LIN {X 104.584,Y 102.598,Z 81.000,A 180.000,B 0.000,C 180.000} C_DIS
LIN {X 104.698,Y 102.438,Z 81.000,A 180.000,B 0.000,C 180.000} C_DIS
LIN {X 104.762,Y 102.341,Z 81.000,A 180.000,B 0.000,C 180.000} C_DIS
LIN {X 104.817,Y 102.260,Z 81.000,A 180.000,B 0.000,C 180.000} C_DIS
LIN {X 104.931,Y 102.081,Z 81.000,A 180.000,B 0.000,C 180.000} C_DIS
LIN {X 105.036,Y 101.902,Z 81.000,A 180.000,B 0.000,C 180.000} C_DIS
LIN {X 105.120,Y 101.755,Z 81.000,A 180.000,B 0.000,C 180.000} C_DIS
LIN {X 105.137,Y 101.723,Z 81.000,A 180.000,B 0.000,C 180.000} C_DIS
LIN {X 105.234,Y 101.545,Z 81.000,A 180.000,B 0.000,C 180.000} C_DIS
LIN {X 105.326,Y 101.366,Z 81.000,A 180.000,B 0.000,C 180.000} C_DIS
LIN {X 105.413,Y 101.187,Z 81.000,A 180.000,B 0.000,C 180.000} C_DIS
LIN {X 105.493,Y 101.008,Z 81.000,A 180.000,B 0.000,C 180.000} C_DIS
LIN {X 105.568,Y 100.829,Z 81.000,A 180.000,B 0.000,C 180.000} C_DIS
LIN {X 105.638,Y 100.651,Z 81.000,A 180.000,B 0.000,C 180.000} C_DIS
LIN {X 105.706,Y 100.472,Z 81.000,A 180.000,B 0.000,C 180.000} C_DIS
LIN {X 105.771,Y 100.293,Z 81.000,A 180.000,B 0.000,C 180.000} C_DIS
LIN {X 105.835,Y 100.092,Z 81.000,A 180.000,B 0.000,C 180.000} C_DIS
LIN {X 105.883,Y 99.936,Z 81.000,A 180.000,B 0.000,C 180.000} C_DIS
LIN {X 105.929,Y 99.757,Z 81.000,A 180.000,B 0.000,C 180.000} C_DIS
LIN {X 105.975,Y 99.578,Z 81.000,A 180.000,B 0.000,C 180.000} C_DIS
LIN {X 106.014,Y 99.427,Z 81.000,A 180.000,B 0.000,C 180.000} C_DIS
LIN {X 106.020,Y 99.399,Z 81.000,A 180.000,B 0.000,C 180.000} C_DIS
LIN {X 106.057,Y 99.221,Z 81.000,A 180.000,B 0.000,C 180.000} C_DIS
LIN {X 106.093,Y 99.042,Z 81.000,A 180.000,B 0.000,C 180.000} C_DIS
LIN {X 106.121,Y 98.863,Z 81.000,A 180.000,B 0.000,C 180.000} C_DIS
LIN {X 106.146,Y 98.684,Z 81.000,A 180.000,B 0.000,C 180.000} C_DIS
LIN {X 106.169,Y 98.505,Z 81.000,A 180.000,B 0.000,C 180.000} C_DIS
LIN {X 106.190,Y 98.327,Z 81.000,A 180.000,B 0.000,C 180.000} C_DIS
LIN {X 106.205,Y 98.148,Z 81.000,A 180.000,B 0.000,C 180.000} C_DIS
LIN {X 106.218,Y 97.969,Z 81.000,A 180.000,B 0.000,C 180.000} C_DIS
LIN {X 106.223,Y 97.790,Z 81.000,A 180.000,B 0.000,C 180.000} C_DIS
LIN {X 106.227,Y 97.612,Z 81.000,A 180.000,B 0.000,C 180.000} C_DIS
LIN {X 106.227,Y 97.433,Z 81.000,A 180.000,B 0.000,C 180.000} C_DIS
LIN {X 106.224,Y 97.254,Z 81.000,A 180.000,B 0.000,C 180.000} C_DIS
LIN {X 106.219,Y 97.075,Z 81.000,A 180.000,B 0.000,C 180.000} C_DIS
LIN {X 106.208,Y 96.897,Z 81.000,A 180.000,B 0.000,C 180.000} C_DIS
LIN {X 106.193,Y 96.709,Z 81.000,A 180.000,B 0.000,C 180.000} C_DIS
LIN {X 106.175,Y 96.539,Z 81.000,A 180.000,B 0.000,C 180.000} C_DIS
LIN {X 106.152,Y 96.360,Z 81.000,A 180.000,B 0.000,C 180.000} C_DIS
LIN {X 106.127,Y 96.181,Z 81.000,A 180.000,B 0.000,C 180.000} C_DIS
LIN {X 106.101,Y 96.003,Z 81.000,A 180.000,B 0.000,C 180.000} C_DIS
LIN {X 106.066,Y 95.824,Z 81.000,A 180.000,B 0.000,C 180.000} C_DIS
LIN {X 106.030,Y 95.645,Z 81.000,A 180.000,B 0.000,C 180.000} C_DIS
LIN {X 106.014,Y 95.573,Z 81.000,A 180.000,B 0.000,C 180.000} C_DIS
LIN {X 105.987,Y 95.466,Z 81.000,A 180.000,B 0.000,C 180.000} C_DIS
LIN {X 105.941,Y 95.288,Z 81.000,A 180.000,B 0.000,C 180.000} C_DIS
LIN {X 105.894,Y 95.109,Z 81.000,A 180.000,B 0.000,C 180.000} C_DIS
LIN {X 105.842,Y 94.930,Z 81.000,A 180.000,B 0.000,C 180.000} C_DIS
LIN {X 105.785,Y 94.751,Z 81.000,A 180.000,B 0.000,C 180.000} C_DIS
LIN {X 105.723,Y 94.573,Z 81.000,A 180.000,B 0.000,C 180.000} C_DIS
LIN {X 105.655,Y 94.394,Z 81.000,A 180.000,B 0.000,C 180.000} C_DIS
LIN {X 105.585,Y 94.215,Z 81.000,A 180.000,B 0.000,C 180.000} C_DIS
LIN {X 105.512,Y 94.036,Z 81.000,A 180.000,B 0.000,C 180.000} C_DIS
LIN {X 105.477,Y 93.958,Z 81.000,A 180.000,B 0.000,C 180.000} C_DIS
LIN {X 105.432,Y 93.857,Z 81.000,A 180.000,B 0.000,C 180.000} C_DIS
LIN {X 105.349,Y 93.679,Z 81.000,A 180.000,B 0.000,C 180.000} C_DIS
LIN {X 105.299,Y 93.581,Z 81.000,A 180.000,B 0.000,C 180.000} C_DIS
LIN {X 105.257,Y 93.500,Z 81.000,A 180.000,B 0.000,C 180.000} C_DIS
LIN {X 105.162,Y 93.321,Z 81.000,A 180.000,B 0.000,C 180.000} C_DIS
LIN {X 105.120,Y 93.245,Z 81.000,A 180.000,B 0.000,C 180.000} C_DIS
LIN {X 105.063,Y 93.142,Z 81.000,A 180.000,B 0.000,C 180.000} C_DIS
LIN {X 104.941,Y 92.936,Z 81.000,A 180.000,B 0.000,C 180.000} C_DIS
LIN {X 104.847,Y 92.785,Z 81.000,A 180.000,B 0.000,C 180.000} C_DIS
LIN {X 104.727,Y 92.606,Z 81.000,A 180.000,B 0.000,C 180.000} C_DIS
LIN {X 104.602,Y 92.427,Z 81.000,A 180.000,B 0.000,C 180.000} C_DIS
LIN {X 104.584,Y 92.402,Z 81.000,A 180.000,B 0.000,C 180.000} C_DIS
LIN {X 104.470,Y 92.249,Z 81.000,A 180.000,B 0.000,C 180.000} C_DIS
LIN {X 104.405,Y 92.162,Z 81.000,A 180.000,B 0.000,C 180.000} C_DIS
LIN {X 104.335,Y 92.070,Z 81.000,A 180.000,B 0.000,C 180.000} C_DIS
LIN {X 104.226,Y 91.936,Z 81.000,A 180.000,B 0.000,C 180.000} C_DIS
LIN {X 104.188,Y 91.891,Z 81.000,A 180.000,B 0.000,C 180.000} C_DIS
LIN {X 104.047,Y 91.726,Z 81.000,A 180.000,B 0.000,C 180.000} C_DIS
LIN {X 104.035,Y 91.712,Z 81.000,A 180.000,B 0.000,C 180.000} C_DIS
LIN {X 103.869,Y 91.535,Z 81.000,A 180.000,B 0.000,C 180.000} C_DIS
LIN {X 103.690,Y 91.346,Z 81.000,A 180.000,B 0.000,C 180.000} C_DIS
LIN {X 103.516,Y 91.176,Z 81.000,A 180.000,B 0.000,C 180.000} C_DIS
LIN {X 103.511,Y 91.171,Z 81.000,A 180.000,B 0.000,C 180.000} C_DIS
LIN {X 103.332,Y 91.004,Z 81.000,A 180.000,B 0.000,C 180.000} C_DIS
LIN {X 103.324,Y 90.997,Z 81.000,A 180.000,B 0.000,C 180.000} C_DIS
LIN {X 103.153,Y 90.852,Z 81.000,A 180.000,B 0.000,C 180.000} C_DIS
LIN {X 103.113,Y 90.818,Z 81.000,A 180.000,B 0.000,C 180.000} C_DIS
LIN {X 102.975,Y 90.703,Z 81.000,A 180.000,B 0.000,C 180.000} C_DIS
LIN {X 102.897,Y 90.640,Z 81.000,A 180.000,B 0.000,C 180.000} C_DIS
LIN {X 102.796,Y 90.562,Z 81.000,A 180.000,B 0.000,C 180.000} C_DIS
LIN {X 102.662,Y 90.461,Z 81.000,A 180.000,B 0.000,C 180.000} C_DIS
LIN {X 102.617,Y 90.427,Z 81.000,A 180.000,B 0.000,C 180.000} C_DIS
LIN {X 102.438,Y 90.303,Z 81.000,A 180.000,B 0.000,C 180.000} C_DIS
LIN {X 102.407,Y 90.282,Z 81.000,A 180.000,B 0.000,C 180.000} C_DIS
LIN {X 102.260,Y 90.184,Z 81.000,A 180.000,B 0.000,C 180.000} C_DIS
LIN {X 102.132,Y 90.103,Z 81.000,A 180.000,B 0.000,C 180.000} C_DIS
LIN {X 102.081,Y 90.071,Z 81.000,A 180.000,B 0.000,C 180.000} C_DIS
LIN {X 101.902,Y 89.963,Z 81.000,A 180.000,B 0.000,C 180.000} C_DIS
LIN {X 101.836,Y 89.925,Z 81.000,A 180.000,B 0.000,C 180.000} C_DIS
LIN {X 101.723,Y 89.859,Z 81.000,A 180.000,B 0.000,C 180.000} C_DIS
LIN {X 101.545,Y 89.765,Z 81.000,A 180.000,B 0.000,C 180.000} C_DIS
LIN {X 101.506,Y 89.746,Z 81.000,A 180.000,B 0.000,C 180.000} C_DIS
LIN {X 101.366,Y 89.674,Z 81.000,A 180.000,B 0.000,C 180.000} C_DIS
LIN {X 101.187,Y 89.590,Z 81.000,A 180.000,B 0.000,C 180.000} C_DIS
LIN {X 101.138,Y 89.567,Z 81.000,A 180.000,B 0.000,C 180.000} C_DIS
LIN {X 101.008,Y 89.509,Z 81.000,A 180.000,B 0.000,C 180.000} C_DIS
LIN {X 100.829,Y 89.430,Z 81.000,A 180.000,B 0.000,C 180.000} C_DIS
LIN {X 100.725,Y 89.388,Z 81.000,A 180.000,B 0.000,C 180.000} C_DIS
LIN {X 100.651,Y 89.360,Z 81.000,A 180.000,B 0.000,C 180.000} C_DIS
LIN {X 100.472,Y 89.292,Z 81.000,A 180.000,B 0.000,C 180.000} C_DIS
LIN {X 100.293,Y 89.232,Z 81.000,A 180.000,B 0.000,C 180.000} C_DIS
LIN {X 100.223,Y 89.209,Z 81.000,A 180.000,B 0.000,C 180.000} C_DIS
LIN {X 100.114,Y 89.175,Z 81.000,A 180.000,B 0.000,C 180.000} C_DIS
LIN {X 99.936,Y 89.118,Z 81.000,A 180.000,B 0.000,C 180.000} C_DIS
LIN {X 99.757,Y 89.068,Z 81.000,A 180.000,B 0.000,C 180.000} C_DIS
LIN {X 99.578,Y 89.022,Z 81.000,A 180.000,B 0.000,C 180.000} C_DIS
LIN {X 99.399,Y 88.981,Z 81.000,A 180.000,B 0.000,C 180.000} C_DIS
LIN {X 99.221,Y 88.945,Z 81.000,A 180.000,B 0.000,C 180.000} C_DIS
LIN {X 99.042,Y 88.910,Z 81.000,A 180.000,B 0.000,C 180.000} C_DIS
LIN {X 98.863,Y 88.878,Z 81.000,A 180.000,B 0.000,C 180.000} C_DIS
LIN {X 98.682,Y 88.852,Z 81.000,A 180.000,B 0.000,C 180.000} C_DIS
LIN {X 98.505,Y 88.828,Z 81.000,A 180.000,B 0.000,C 180.000} C_DIS
LIN {X 98.327,Y 88.811,Z 81.000,A 180.000,B 0.000,C 180.000} C_DIS
LIN {X 98.148,Y 88.796,Z 81.000,A 180.000,B 0.000,C 180.000} C_DIS
LIN {X 97.969,Y 88.785,Z 81.000,A 180.000,B 0.000,C 180.000} C_DIS
LIN {X 97.790,Y 88.777,Z 81.000,A 180.000,B 0.000,C 180.000} C_DIS
LIN {X 97.612,Y 88.772,Z 81.000,A 180.000,B 0.000,C 180.000} C_DIS
LIN {X 97.433,Y 88.770,Z 81.000,A 180.000,B 0.000,C 180.000} C_DIS
LIN {X 97.254,Y 88.775,Z 81.000,A 180.000,B 0.000,C 180.000} C_DIS
LIN {X 97.075,Y 88.782,Z 81.000,A 180.000,B 0.000,C 180.000} C_DIS
LIN {X 96.897,Y 88.793,Z 81.000,A 180.000,B 0.000,C 180.000} C_DIS
LIN {X 96.718,Y 88.808,Z 81.000,A 180.000,B 0.000,C 180.000} C_DIS
LIN {X 96.539,Y 88.823,Z 81.000,A 180.000,B 0.000,C 180.000} C_DIS
LIN {X 96.360,Y 88.846,Z 81.000,A 180.000,B 0.000,C 180.000} C_DIS
LIN {X 96.181,Y 88.871,Z 81.000,A 180.000,B 0.000,C 180.000} C_DIS
LIN {X 96.003,Y 88.902,Z 81.000,A 180.000,B 0.000,C 180.000} C_DIS
LIN {X 95.824,Y 88.936,Z 81.000,A 180.000,B 0.000,C 180.000} C_DIS
LIN {X 95.645,Y 88.972,Z 81.000,A 180.000,B 0.000,C 180.000} C_DIS
LIN {X 95.466,Y 89.010,Z 81.000,A 180.000,B 0.000,C 180.000} C_DIS
LIN {X 95.387,Y 89.031,Z 81.000,A 180.000,B 0.000,C 180.000} C_DIS
LIN {X 95.288,Y 89.056,Z 81.000,A 180.000,B 0.000,C 180.000} C_DIS
LIN {X 95.109,Y 89.104,Z 81.000,A 180.000,B 0.000,C 180.000} C_DIS
LIN {X 94.930,Y 89.161,Z 81.000,A 180.000,B 0.000,C 180.000} C_DIS
LIN {X 94.777,Y 89.209,Z 81.000,A 180.000,B 0.000,C 180.000} C_DIS
LIN {X 94.751,Y 89.218,Z 81.000,A 180.000,B 0.000,C 180.000} C_DIS
LIN {X 94.573,Y 89.276,Z 81.000,A 180.000,B 0.000,C 180.000} C_DIS
LIN {X 94.394,Y 89.343,Z 81.000,A 180.000,B 0.000,C 180.000} C_DIS
LIN {X 94.275,Y 89.388,Z 81.000,A 180.000,B 0.000,C 180.000} C_DIS
LIN {X 94.215,Y 89.411,Z 81.000,A 180.000,B 0.000,C 180.000} C_DIS
LIN {X 94.036,Y 89.489,Z 81.000,A 180.000,B 0.000,C 180.000} C_DIS
LIN {X 93.862,Y 89.567,Z 81.000,A 180.000,B 0.000,C 180.000} C_DIS
LIN {X 93.857,Y 89.569,Z 81.000,A 180.000,B 0.000,C 180.000} C_DIS
LIN {X 93.679,Y 89.653,Z 81.000,A 180.000,B 0.000,C 180.000} C_DIS
LIN {X 93.500,Y 89.742,Z 81.000,A 180.000,B 0.000,C 180.000} C_DIS
LIN {X 93.321,Y 89.835,Z 81.000,A 180.000,B 0.000,C 180.000} C_DIS
LIN {X 93.164,Y 89.925,Z 81.000,A 180.000,B 0.000,C 180.000} C_DIS
LIN {X 93.142,Y 89.937,Z 81.000,A 180.000,B 0.000,C 180.000} C_DIS
LIN {X 92.964,Y 90.043,Z 81.000,A 180.000,B 0.000,C 180.000} C_DIS
LIN {X 92.868,Y 90.103,Z 81.000,A 180.000,B 0.000,C 180.000} C_DIS
LIN {X 92.785,Y 90.156,Z 81.000,A 180.000,B 0.000,C 180.000} C_DIS
LIN {X 92.606,Y 90.274,Z 81.000,A 180.000,B 0.000,C 180.000} C_DIS
LIN {X 92.593,Y 90.282,Z 81.000,A 180.000,B 0.000,C 180.000} C_DIS
LIN {X 92.427,Y 90.395,Z 81.000,A 180.000,B 0.000,C 180.000} C_DIS
LIN {X 92.338,Y 90.461,Z 81.000,A 180.000,B 0.000,C 180.000} C_DIS
LIN {X 92.249,Y 90.528,Z 81.000,A 180.000,B 0.000,C 180.000} C_DIS
LIN {X 92.103,Y 90.640,Z 81.000,A 180.000,B 0.000,C 180.000} C_DIS
LIN {X 92.070,Y 90.667,Z 81.000,A 180.000,B 0.000,C 180.000} C_DIS
LIN {X 91.891,Y 90.815,Z 81.000,A 180.000,B 0.000,C 180.000} C_DIS
LIN {X 91.712,Y 90.966,Z 81.000,A 180.000,B 0.000,C 180.000} C_DIS
LIN {X 91.676,Y 90.997,Z 81.000,A 180.000,B 0.000,C 180.000} C_DIS
LIN {X 91.533,Y 91.129,Z 81.000,A 180.000,B 0.000,C 180.000} C_DIS
LIN {X 91.484,Y 91.176,Z 81.000,A 180.000,B 0.000,C 180.000} C_DIS
LIN {X 91.355,Y 91.300,Z 81.000,A 180.000,B 0.000,C 180.000} C_DIS
LIN {X 91.302,Y 91.355,Z 81.000,A 180.000,B 0.000,C 180.000} C_DIS
LIN {X 91.133,Y 91.533,Z 81.000,A 180.000,B 0.000,C 180.000} C_DIS
LIN {X 90.997,Y 91.678,Z 81.000,A 180.000,B 0.000,C 180.000} C_DIS
LIN {X 90.965,Y 91.712,Z 81.000,A 180.000,B 0.000,C 180.000} C_DIS
LIN {X 90.818,Y 91.884,Z 81.000,A 180.000,B 0.000,C 180.000} C_DIS
LIN {X 90.812,Y 91.891,Z 81.000,A 180.000,B 0.000,C 180.000} C_DIS
LIN {X 90.665,Y 92.070,Z 81.000,A 180.000,B 0.000,C 180.000} C_DIS
LIN {X 90.640,Y 92.103,Z 81.000,A 180.000,B 0.000,C 180.000} C_DIS
LIN {X 90.530,Y 92.249,Z 81.000,A 180.000,B 0.000,C 180.000} C_DIS
LIN {X 90.461,Y 92.341,Z 81.000,A 180.000,B 0.000,C 180.000} C_DIS
LIN {X 90.398,Y 92.427,Z 81.000,A 180.000,B 0.000,C 180.000} C_DIS
LIN {X 90.282,Y 92.592,Z 81.000,A 180.000,B 0.000,C 180.000} C_DIS
LIN {X 90.153,Y 92.785,Z 81.000,A 180.000,B 0.000,C 180.000} C_DIS
LIN {X 90.103,Y 92.862,Z 81.000,A 180.000,B 0.000,C 180.000} C_DIS
LIN {X 90.082,Y 92.898,Z 81.000,A 180.000,B 0.000,C 180.000} C_DIS
; Link Move Starts
LIN {X 89.924,Y 93.166,Z 81.000,A 180.000,B 0.000,C 180.000} C_DIS
LIN {X 89.783,Y 93.422,Z 80.999,A 180.000,B 0.000,C 180.000} C_DIS
LIN {X 89.639,Y 93.700,Z 80.998,A 180.000,B 0.000,C 180.000} C_DIS
LIN {X 89.518,Y 93.964,Z 80.996,A 180.000,B 0.000,C 180.000} C_DIS
LIN {X 89.405,Y 94.233,Z 80.995,A 180.000,B 0.000,C 180.000} C_DIS
LIN {X 89.292,Y 94.523,Z 80.992,A 180.000,B 0.000,C 180.000} C_DIS
LIN {X 89.195,Y 94.796,Z 80.989,A 180.000,B 0.000,C 180.000} C_DIS
LIN {X 89.108,Y 95.073,Z 80.986,A 180.000,B 0.000,C 180.000} C_DIS
LIN {X 89.028,Y 95.376,Z 80.983,A 180.000,B 0.000,C 180.000} C_DIS
LIN {X 88.956,Y 95.663,Z 80.979,A 180.000,B 0.000,C 180.000} C_DIS
LIN {X 88.896,Y 95.955,Z 80.974,A 180.000,B 0.000,C 180.000} C_DIS
LIN {X 88.849,Y 96.249,Z 80.970,A 180.000,B 0.000,C 180.000} C_DIS
LIN {X 88.827,Y 96.403,Z 80.967,A 180.000,B 0.000,C 180.000} C_DIS
LIN {X 88.806,Y 96.556,Z 80.965,A 180.000,B 0.000,C 180.000} C_DIS
LIN {X 88.790,Y 96.704,Z 80.962,A 180.000,B 0.000,C 180.000} C_DIS
LIN {X 88.776,Y 96.852,Z 80.959,A 180.000,B 0.000,C 180.000} C_DIS
LIN {X 88.764,Y 96.996,Z 80.957,A 180.000,B 0.000,C 180.000} C_DIS
LIN {X 88.757,Y 97.141,Z 80.954,A 180.000,B 0.000,C 180.000} C_DIS
LIN {X 88.752,Y 97.292,Z 80.951,A 180.000,B 0.000,C 180.000} C_DIS
LIN {X 88.748,Y 97.443,Z 80.948,A 180.000,B 0.000,C 180.000} C_DIS
LIN {X 88.747,Y 97.595,Z 80.944,A 180.000,B 0.000,C 180.000} C_DIS
LIN {X 88.748,Y 97.747,Z 80.941,A 180.000,B 0.000,C 180.000} C_DIS
LIN {X 88.751,Y 97.896,Z 80.938,A 180.000,B 0.000,C 180.000} C_DIS
LIN {X 88.756,Y 98.044,Z 80.934,A 180.000,B 0.000,C 180.000} C_DIS
LIN {X 88.767,Y 98.194,Z 80.931,A 180.000,B 0.000,C 180.000} C_DIS
LIN {X 88.778,Y 98.344,Z 80.927,A 180.000,B 0.000,C 180.000} C_DIS
LIN {X 88.793,Y 98.492,Z 80.924,A 180.000,B 0.000,C 180.000} C_DIS
LIN {X 88.810,Y 98.640,Z 80.920,A 180.000,B 0.000,C 180.000} C_DIS
LIN {X 88.830,Y 98.796,Z 80.916,A 180.000,B 0.000,C 180.000} C_DIS
LIN {X 88.850,Y 98.951,Z 80.912,A 180.000,B 0.000,C 180.000} C_DIS
LIN {X 88.874,Y 99.095,Z 80.908,A 180.000,B 0.000,C 180.000} C_DIS
LIN {X 88.901,Y 99.239,Z 80.904,A 180.000,B 0.000,C 180.000} C_DIS
LIN {X 88.928,Y 99.382,Z 80.900,A 180.000,B 0.000,C 180.000} C_DIS
LIN {X 88.961,Y 99.525,Z 80.896,A 180.000,B 0.000,C 180.000} C_DIS
LIN {X 88.998,Y 99.677,Z 80.892,A 180.000,B 0.000,C 180.000} C_DIS
LIN {X 89.036,Y 99.830,Z 80.888,A 180.000,B 0.000,C 180.000} C_DIS
LIN {X 89.071,Y 99.972,Z 80.883,A 180.000,B 0.000,C 180.000} C_DIS
LIN {X 89.112,Y 100.113,Z 80.879,A 180.000,B 0.000,C 180.000} C_DIS
LIN {X 89.156,Y 100.255,Z 80.875,A 180.000,B 0.000,C 180.000} C_DIS
LIN {X 89.200,Y 100.397,Z 80.870,A 180.000,B 0.000,C 180.000} C_DIS
LIN {X 89.253,Y 100.541,Z 80.865,A 180.000,B 0.000,C 180.000} C_DIS
LIN {X 89.305,Y 100.685,Z 80.861,A 180.000,B 0.000,C 180.000} C_DIS
LIN {X 89.358,Y 100.824,Z 80.856,A 180.000,B 0.000,C 180.000} C_DIS
LIN {X 89.412,Y 100.964,Z 80.851,A 180.000,B 0.000,C 180.000} C_DIS
LIN {X 89.473,Y 101.106,Z 80.846,A 180.000,B 0.000,C 180.000} C_DIS
LIN {X 89.503,Y 101.176,Z 80.844,A 180.000,B 0.000,C 180.000} C_DIS
LIN {X 89.533,Y 101.247,Z 80.841,A 180.000,B 0.000,C 180.000} C_DIS
LIN {X 89.596,Y 101.381,Z 80.836,A 180.000,B 0.000,C 180.000} C_DIS
LIN {X 89.662,Y 101.514,Z 80.831,A 180.000,B 0.000,C 180.000} C_DIS
LIN {X 89.696,Y 101.582,Z 80.829,A 180.000,B 0.000,C 180.000} C_DIS
LIN {X 89.730,Y 101.650,Z 80.826,A 180.000,B 0.000,C 180.000} C_DIS
LIN {X 89.765,Y 101.717,Z 80.824,A 180.000,B 0.000,C 180.000} C_DIS
LIN {X 89.801,Y 101.784,Z 80.821,A 180.000,B 0.000,C 180.000} C_DIS
LIN {X 89.836,Y 101.851,Z 80.818,A 180.000,B 0.000,C 180.000} C_DIS
LIN {X 89.873,Y 101.918,Z 80.816,A 180.000,B 0.000,C 180.000} C_DIS
LIN {X 89.949,Y 102.051,Z 80.811,A 180.000,B 0.000,C 180.000} C_DIS
LIN {X 89.985,Y 102.115,Z 80.808,A 180.000,B 0.000,C 180.000} C_DIS
LIN {X 90.022,Y 102.178,Z 80.805,A 180.000,B 0.000,C 180.000} C_DIS
LIN {X 90.060,Y 102.241,Z 80.803,A 180.000,B 0.000,C 180.000} C_DIS
LIN {X 90.100,Y 102.303,Z 80.800,A 180.000,B 0.000,C 180.000} C_DIS
LIN {X 90.183,Y 102.431,Z 80.795,A 180.000,B 0.000,C 180.000} C_DIS
LIN {X 90.224,Y 102.496,Z 80.792,A 180.000,B 0.000,C 180.000} C_DIS
LIN {X 90.267,Y 102.559,Z 80.790,A 180.000,B 0.000,C 180.000} C_DIS
LIN {X 90.354,Y 102.683,Z 80.784,A 180.000,B 0.000,C 180.000} C_DIS
LIN {X 90.398,Y 102.745,Z 80.782,A 180.000,B 0.000,C 180.000} C_DIS
LIN {X 90.443,Y 102.807,Z 80.779,A 180.000,B 0.000,C 180.000} C_DIS
LIN {X 90.532,Y 102.929,Z 80.774,A 180.000,B 0.000,C 180.000} C_DIS
LIN {X 90.576,Y 102.991,Z 80.771,A 180.000,B 0.000,C 180.000} C_DIS
LIN {X 90.622,Y 103.051,Z 80.768,A 180.000,B 0.000,C 180.000} C_DIS
LIN {X 90.669,Y 103.109,Z 80.766,A 180.000,B 0.000,C 180.000} C_DIS
LIN {X 90.764,Y 103.225,Z 80.761,A 180.000,B 0.000,C 180.000} C_DIS
LIN {X 90.812,Y 103.283,Z 80.758,A 180.000,B 0.000,C 180.000} C_DIS
LIN {X 90.860,Y 103.342,Z 80.755,A 180.000,B 0.000,C 180.000} C_DIS
LIN {X 90.910,Y 103.398,Z 80.753,A 180.000,B 0.000,C 180.000} C_DIS
LIN {X 91.012,Y 103.510,Z 80.747,A 180.000,B 0.000,C 180.000} C_DIS
LIN {X 91.065,Y 103.568,Z 80.745,A 180.000,B 0.000,C 180.000} C_DIS
LIN {X 91.171,Y 103.684,Z 80.739,A 180.000,B 0.000,C 180.000} C_DIS
LIN {X 91.224,Y 103.742,Z 80.736,A 180.000,B 0.000,C 180.000} C_DIS
LIN {X 91.275,Y 103.796,Z 80.734,A 180.000,B 0.000,C 180.000} C_DIS
LIN {X 91.327,Y 103.848,Z 80.731,A 180.000,B 0.000,C 180.000} C_DIS
LIN {X 91.486,Y 104.004,Z 80.724,A 180.000,B 0.000,C 180.000} C_DIS
LIN {X 91.539,Y 104.055,Z 80.721,A 180.000,B 0.000,C 180.000} C_DIS
LIN {X 91.594,Y 104.106,Z 80.718,A 180.000,B 0.000,C 180.000} C_DIS
LIN {X 91.649,Y 104.154,Z 80.716,A 180.000,B 0.000,C 180.000} C_DIS
LIN {X 91.767,Y 104.257,Z 80.710,A 180.000,B 0.000,C 180.000} C_DIS
LIN {X 91.825,Y 104.308,Z 80.708,A 180.000,B 0.000,C 180.000} C_DIS
LIN {X 91.884,Y 104.359,Z 80.705,A 180.000,B 0.000,C 180.000} C_DIS
LIN {X 91.942,Y 104.408,Z 80.702,A 180.000,B 0.000,C 180.000} C_DIS
LIN {X 91.999,Y 104.456,Z 80.700,A 180.000,B 0.000,C 180.000} C_DIS
LIN {X 92.057,Y 104.504,Z 80.697,A 180.000,B 0.000,C 180.000} C_DIS
LIN {X 92.116,Y 104.550,Z 80.694,A 180.000,B 0.000,C 180.000} C_DIS
LIN {X 92.236,Y 104.644,Z 80.689,A 180.000,B 0.000,C 180.000} C_DIS
LIN {X 92.296,Y 104.691,Z 80.686,A 180.000,B 0.000,C 180.000} C_DIS
LIN {X 92.357,Y 104.737,Z 80.684,A 180.000,B 0.000,C 180.000} C_DIS
LIN {X 92.419,Y 104.780,Z 80.681,A 180.000,B 0.000,C 180.000} C_DIS
LIN {X 92.543,Y 104.866,Z 80.676,A 180.000,B 0.000,C 180.000} C_DIS
LIN {X 92.605,Y 104.909,Z 80.673,A 180.000,B 0.000,C 180.000} C_DIS
LIN {X 92.669,Y 104.953,Z 80.670,A 180.000,B 0.000,C 180.000} C_DIS
LIN {X 92.733,Y 104.995,Z 80.668,A 180.000,B 0.000,C 180.000} C_DIS
LIN {X 92.797,Y 105.037,Z 80.665,A 180.000,B 0.000,C 180.000} C_DIS
LIN {X 92.861,Y 105.079,Z 80.662,A 180.000,B 0.000,C 180.000} C_DIS
LIN {X 92.925,Y 105.119,Z 80.660,A 180.000,B 0.000,C 180.000} C_DIS
LIN {X 93.119,Y 105.237,Z 80.652,A 180.000,B 0.000,C 180.000} C_DIS
LIN {X 93.184,Y 105.277,Z 80.649,A 180.000,B 0.000,C 180.000} C_DIS
LIN {X 93.251,Y 105.314,Z 80.647,A 180.000,B 0.000,C 180.000} C_DIS
LIN {X 93.318,Y 105.351,Z 80.644,A 180.000,B 0.000,C 180.000} C_DIS
LIN {X 93.453,Y 105.423,Z 80.639,A 180.000,B 0.000,C 180.000} C_DIS
LIN {X 93.520,Y 105.459,Z 80.636,A 180.000,B 0.000,C 180.000} C_DIS
LIN {X 93.588,Y 105.493,Z 80.633,A 180.000,B 0.000,C 180.000} C_DIS
LIN {X 93.725,Y 105.561,Z 80.628,A 180.000,B 0.000,C 180.000} C_DIS
LIN {X 93.795,Y 105.595,Z 80.625,A 180.000,B 0.000,C 180.000} C_DIS
LIN {X 94.003,Y 105.692,Z 80.617,A 180.000,B 0.000,C 180.000} C_DIS
LIN {X 94.071,Y 105.723,Z 80.615,A 180.000,B 0.000,C 180.000} C_DIS
LIN {X 94.139,Y 105.753,Z 80.612,A 180.000,B 0.000,C 180.000} C_DIS
LIN {X 94.209,Y 105.781,Z 80.609,A 180.000,B 0.000,C 180.000} C_DIS
LIN {X 94.420,Y 105.866,Z 80.601,A 180.000,B 0.000,C 180.000} C_DIS
LIN {X 94.491,Y 105.893,Z 80.599,A 180.000,B 0.000,C 180.000} C_DIS
LIN {X 94.564,Y 105.919,Z 80.596,A 180.000,B 0.000,C 180.000} C_DIS
LIN {X 94.711,Y 105.970,Z 80.591,A 180.000,B 0.000,C 180.000} C_DIS
LIN {X 94.785,Y 105.995,Z 80.588,A 180.000,B 0.000,C 180.000} C_DIS
LIN {X 95.002,Y 106.068,Z 80.580,A 180.000,B 0.000,C 180.000} C_DIS
LIN {X 95.075,Y 106.091,Z 80.577,A 180.000,B 0.000,C 180.000} C_DIS
LIN {X 95.148,Y 106.113,Z 80.574,A 180.000,B 0.000,C 180.000} C_DIS
LIN {X 95.368,Y 106.173,Z 80.567,A 180.000,B 0.000,C 180.000} C_DIS
LIN {X 95.442,Y 106.193,Z 80.564,A 180.000,B 0.000,C 180.000} C_DIS
LIN {X 95.516,Y 106.211,Z 80.561,A 180.000,B 0.000,C 180.000} C_DIS
LIN {X 95.590,Y 106.227,Z 80.559,A 180.000,B 0.000,C 180.000} C_DIS
LIN {X 95.817,Y 106.276,Z 80.550,A 180.000,B 0.000,C 180.000} C_DIS
LIN {X 95.894,Y 106.292,Z 80.548,A 180.000,B 0.000,C 180.000} C_DIS
LIN {X 95.970,Y 106.308,Z 80.545,A 180.000,B 0.000,C 180.000} C_DIS
LIN {X 96.045,Y 106.323,Z 80.542,A 180.000,B 0.000,C 180.000} C_DIS
LIN {X 96.119,Y 106.337,Z 80.540,A 180.000,B 0.000,C 180.000} C_DIS
LIN {X 96.194,Y 106.349,Z 80.537,A 180.000,B 0.000,C 180.000} C_DIS
LIN {X 96.343,Y 106.372,Z 80.532,A 180.000,B 0.000,C 180.000} C_DIS
LIN {X 96.418,Y 106.384,Z 80.529,A 180.000,B 0.000,C 180.000} C_DIS
LIN {X 96.493,Y 106.394,Z 80.526,A 180.000,B 0.000,C 180.000} C_DIS
LIN {X 96.567,Y 106.402,Z 80.524,A 180.000,B 0.000,C 180.000} C_DIS
LIN {X 96.801,Y 106.426,Z 80.516,A 180.000,B 0.000,C 180.000} C_DIS
LIN {X 96.879,Y 106.433,Z 80.513,A 180.000,B 0.000,C 180.000} C_DIS
LIN {X 97.031,Y 106.445,Z 80.508,A 180.000,B 0.000,C 180.000} C_DIS
LIN {X 97.107,Y 106.451,Z 80.505,A 180.000,B 0.000,C 180.000} C_DIS
LIN {X 97.183,Y 106.455,Z 80.502,A 180.000,B 0.000,C 180.000} C_DIS
LIN {X 97.412,Y 106.465,Z 80.494,A 180.000,B 0.000,C 180.000} C_DIS
LIN {X 97.489,Y 106.468,Z 80.492,A 180.000,B 0.000,C 180.000} C_DIS
LIN {X 97.566,Y 106.468,Z 80.489,A 180.000,B 0.000,C 180.000} C_DIS
LIN {X 97.796,Y 106.465,Z 80.481,A 180.000,B 0.000,C 180.000} C_DIS
LIN {X 97.874,Y 106.464,Z 80.478,A 180.000,B 0.000,C 180.000} C_DIS
LIN {X 97.951,Y 106.461,Z 80.475,A 180.000,B 0.000,C 180.000} C_DIS
LIN {X 98.106,Y 106.454,Z 80.470,A 180.000,B 0.000,C 180.000} C_DIS
LIN {X 98.183,Y 106.450,Z 80.467,A 180.000,B 0.000,C 180.000} C_DIS
LIN {X 98.415,Y 106.434,Z 80.459,A 180.000,B 0.000,C 180.000} C_DIS
LIN {X 98.491,Y 106.429,Z 80.457,A 180.000,B 0.000,C 180.000} C_DIS
LIN {X 98.567,Y 106.421,Z 80.454,A 180.000,B 0.000,C 180.000} C_DIS
LIN {X 98.642,Y 106.412,Z 80.451,A 180.000,B 0.000,C 180.000} C_DIS
LIN {X 98.868,Y 106.384,Z 80.443,A 180.000,B 0.000,C 180.000} C_DIS
LIN {X 98.944,Y 106.373,Z 80.441,A 180.000,B 0.000,C 180.000} C_DIS
LIN {X 99.019,Y 106.361,Z 80.438,A 180.000,B 0.000,C 180.000} C_DIS
LIN {X 99.174,Y 106.334,Z 80.432,A 180.000,B 0.000,C 180.000} C_DIS
LIN {X 99.251,Y 106.320,Z 80.430,A 180.000,B 0.000,C 180.000} C_DIS
LIN {X 99.478,Y 106.279,Z 80.422,A 180.000,B 0.000,C 180.000} C_DIS
LIN {X 99.553,Y 106.264,Z 80.419,A 180.000,B 0.000,C 180.000} C_DIS
LIN {X 99.627,Y 106.247,Z 80.416,A 180.000,B 0.000,C 180.000} C_DIS
LIN {X 99.851,Y 106.193,Z 80.408,A 180.000,B 0.000,C 180.000} C_DIS
LIN {X 99.926,Y 106.174,Z 80.406,A 180.000,B 0.000,C 180.000} C_DIS
LIN {X 100.001,Y 106.154,Z 80.403,A 180.000,B 0.000,C 180.000} C_DIS
LIN {X 100.075,Y 106.131,Z 80.400,A 180.000,B 0.000,C 180.000} C_DIS
LIN {X 100.224,Y 106.086,Z 80.395,A 180.000,B 0.000,C 180.000} C_DIS
LIN {X 100.299,Y 106.064,Z 80.392,A 180.000,B 0.000,C 180.000} C_DIS
LIN {X 100.447,Y 106.018,Z 80.387,A 180.000,B 0.000,C 180.000} C_DIS
LIN {X 100.522,Y 105.995,Z 80.384,A 180.000,B 0.000,C 180.000} C_DIS
LIN {X 100.595,Y 105.970,Z 80.381,A 180.000,B 0.000,C 180.000} C_DIS
LIN {X 100.740,Y 105.918,Z 80.376,A 180.000,B 0.000,C 180.000} C_DIS
LIN {X 100.812,Y 105.891,Z 80.373,A 180.000,B 0.000,C 180.000} C_DIS
LIN {X 100.884,Y 105.865,Z 80.370,A 180.000,B 0.000,C 180.000} C_DIS
LIN {X 100.956,Y 105.837,Z 80.368,A 180.000,B 0.000,C 180.000} C_DIS
LIN {X 101.026,Y 105.807,Z 80.365,A 180.000,B 0.000,C 180.000} C_DIS
LIN {X 101.168,Y 105.747,Z 80.360,A 180.000,B 0.000,C 180.000} C_DIS
LIN {X 101.240,Y 105.716,Z 80.357,A 180.000,B 0.000,C 180.000} C_DIS
LIN {X 101.311,Y 105.685,Z 80.354,A 180.000,B 0.000,C 180.000} C_DIS
LIN {X 101.452,Y 105.621,Z 80.349,A 180.000,B 0.000,C 180.000} C_DIS
LIN {X 101.522,Y 105.589,Z 80.346,A 180.000,B 0.000,C 180.000} C_DIS
LIN {X 101.592,Y 105.555,Z 80.343,A 180.000,B 0.000,C 180.000} C_DIS
LIN {X 101.661,Y 105.520,Z 80.341,A 180.000,B 0.000,C 180.000} C_DIS
LIN {X 101.799,Y 105.452,Z 80.335,A 180.000,B 0.000,C 180.000} C_DIS
LIN {X 101.868,Y 105.417,Z 80.333,A 180.000,B 0.000,C 180.000} C_DIS
LIN {X 101.936,Y 105.379,Z 80.330,A 180.000,B 0.000,C 180.000} C_DIS
LIN {X 102.070,Y 105.303,Z 80.325,A 180.000,B 0.000,C 180.000} C_DIS
LIN {X 102.137,Y 105.265,Z 80.322,A 180.000,B 0.000,C 180.000} C_DIS
LIN {X 102.205,Y 105.226,Z 80.319,A 180.000,B 0.000,C 180.000} C_DIS
LIN {X 102.271,Y 105.186,Z 80.316,A 180.000,B 0.000,C 180.000} C_DIS
LIN {X 102.404,Y 105.105,Z 80.311,A 180.000,B 0.000,C 180.000} C_DIS
LIN {X 102.470,Y 105.063,Z 80.308,A 180.000,B 0.000,C 180.000} C_DIS
LIN {X 102.600,Y 104.980,Z 80.303,A 180.000,B 0.000,C 180.000} C_DIS
LIN {X 102.665,Y 104.938,Z 80.300,A 180.000,B 0.000,C 180.000} C_DIS
LIN {X 102.729,Y 104.896,Z 80.298,A 180.000,B 0.000,C 180.000} C_DIS
LIN {X 102.794,Y 104.851,Z 80.295,A 180.000,B 0.000,C 180.000} C_DIS
LIN {X 102.857,Y 104.806,Z 80.292,A 180.000,B 0.000,C 180.000} C_DIS
LIN {X 103.046,Y 104.668,Z 80.284,A 180.000,B 0.000,C 180.000} C_DIS
LIN {X 103.107,Y 104.622,Z 80.281,A 180.000,B 0.000,C 180.000} C_DIS
LIN {X 103.168,Y 104.573,Z 80.279,A 180.000,B 0.000,C 180.000} C_DIS
LIN {X 103.229,Y 104.525,Z 80.276,A 180.000,B 0.000,C 180.000} C_DIS
LIN {X 103.290,Y 104.476,Z 80.273,A 180.000,B 0.000,C 180.000} C_DIS
LIN {X 103.350,Y 104.427,Z 80.270,A 180.000,B 0.000,C 180.000} C_DIS
LIN {X 103.471,Y 104.328,Z 80.265,A 180.000,B 0.000,C 180.000} C_DIS
LIN {X 103.531,Y 104.279,Z 80.262,A 180.000,B 0.000,C 180.000} C_DIS
LIN {X 103.590,Y 104.229,Z 80.259,A 180.000,B 0.000,C 180.000} C_DIS
LIN {X 103.647,Y 104.177,Z 80.257,A 180.000,B 0.000,C 180.000} C_DIS
LIN {X 103.704,Y 104.125,Z 80.254,A 180.000,B 0.000,C 180.000} C_DIS
LIN {X 103.818,Y 104.021,Z 80.249,A 180.000,B 0.000,C 180.000} C_DIS
LIN {X 103.875,Y 103.968,Z 80.246,A 180.000,B 0.000,C 180.000} C_DIS
LIN {X 103.930,Y 103.914,Z 80.243,A 180.000,B 0.000,C 180.000} C_DIS
LIN {X 103.985,Y 103.858,Z 80.241,A 180.000,B 0.000,C 180.000} C_DIS
LIN {X 104.094,Y 103.745,Z 80.235,A 180.000,B 0.000,C 180.000} C_DIS
LIN {X 104.149,Y 103.689,Z 80.232,A 180.000,B 0.000,C 180.000} C_DIS
LIN {X 104.257,Y 103.578,Z 80.227,A 180.000,B 0.000,C 180.000} C_DIS
LIN {X 104.311,Y 103.522,Z 80.224,A 180.000,B 0.000,C 180.000} C_DIS
LIN {X 104.363,Y 103.464,Z 80.222,A 180.000,B 0.000,C 180.000} C_DIS
LIN {X 104.465,Y 103.347,Z 80.216,A 180.000,B 0.000,C 180.000} C_DIS
LIN {X 104.516,Y 103.288,Z 80.213,A 180.000,B 0.000,C 180.000} C_DIS
LIN {X 104.567,Y 103.230,Z 80.211,A 180.000,B 0.000,C 180.000} C_DIS
LIN {X 104.617,Y 103.170,Z 80.208,A 180.000,B 0.000,C 180.000} C_DIS
LIN {X 104.665,Y 103.108,Z 80.205,A 180.000,B 0.000,C 180.000} C_DIS
LIN {X 104.809,Y 102.923,Z 80.197,A 180.000,B 0.000,C 180.000} C_DIS
LIN {X 104.856,Y 102.862,Z 80.194,A 180.000,B 0.000,C 180.000} C_DIS
LIN {X 104.950,Y 102.737,Z 80.189,A 180.000,B 0.000,C 180.000} C_DIS
LIN {X 104.996,Y 102.674,Z 80.186,A 180.000,B 0.000,C 180.000} C_DIS
LIN {X 105.041,Y 102.609,Z 80.183,A 180.000,B 0.000,C 180.000} C_DIS
LIN {X 105.086,Y 102.545,Z 80.181,A 180.000,B 0.000,C 180.000} C_DIS
LIN {X 105.130,Y 102.480,Z 80.178,A 180.000,B 0.000,C 180.000} C_DIS
LIN {X 105.174,Y 102.416,Z 80.176,A 180.000,B 0.000,C 180.000} C_DIS
LIN {X 105.218,Y 102.352,Z 80.173,A 180.000,B 0.000,C 180.000} C_DIS
LIN {X 105.259,Y 102.286,Z 80.170,A 180.000,B 0.000,C 180.000} C_DIS
LIN {X 105.340,Y 102.153,Z 80.165,A 180.000,B 0.000,C 180.000} C_DIS
LIN {X 105.381,Y 102.086,Z 80.163,A 180.000,B 0.000,C 180.000} C_DIS
LIN {X 105.422,Y 102.019,Z 80.160,A 180.000,B 0.000,C 180.000} C_DIS
LIN {X 105.461,Y 101.952,Z 80.157,A 180.000,B 0.000,C 180.000} C_DIS
LIN {X 105.499,Y 101.884,Z 80.155,A 180.000,B 0.000,C 180.000} C_DIS
LIN {X 105.538,Y 101.816,Z 80.152,A 180.000,B 0.000,C 180.000} C_DIS
LIN {X 105.612,Y 101.678,Z 80.147,A 180.000,B 0.000,C 180.000} C_DIS
LIN {X 105.686,Y 101.540,Z 80.143,A 180.000,B 0.000,C 180.000} C_DIS
LIN {X 105.757,Y 101.401,Z 80.138,A 180.000,B 0.000,C 180.000} C_DIS
LIN {X 105.823,Y 101.259,Z 80.133,A 180.000,B 0.000,C 180.000} C_DIS
LIN {X 105.889,Y 101.117,Z 80.128,A 180.000,B 0.000,C 180.000} C_DIS
LIN {X 105.950,Y 100.973,Z 80.124,A 180.000,B 0.000,C 180.000} C_DIS
LIN {X 106.010,Y 100.828,Z 80.119,A 180.000,B 0.000,C 180.000} C_DIS
LIN {X 106.068,Y 100.682,Z 80.114,A 180.000,B 0.000,C 180.000} C_DIS
LIN {X 106.126,Y 100.536,Z 80.110,A 180.000,B 0.000,C 180.000} C_DIS
LIN {X 106.178,Y 100.389,Z 80.106,A 180.000,B 0.000,C 180.000} C_DIS
LIN {X 106.227,Y 100.241,Z 80.101,A 180.000,B 0.000,C 180.000} C_DIS
LIN {X 106.276,Y 100.092,Z 80.097,A 180.000,B 0.000,C 180.000} C_DIS
LIN {X 106.318,Y 99.941,Z 80.093,A 180.000,B 0.000,C 180.000} C_DIS
LIN {X 106.359,Y 99.790,Z 80.089,A 180.000,B 0.000,C 180.000} C_DIS
LIN {X 106.400,Y 99.638,Z 80.085,A 180.000,B 0.000,C 180.000} C_DIS
LIN {X 106.440,Y 99.486,Z 80.081,A 180.000,B 0.000,C 180.000} C_DIS
LIN {X 106.474,Y 99.333,Z 80.077,A 180.000,B 0.000,C 180.000} C_DIS
LIN {X 106.506,Y 99.180,Z 80.073,A 180.000,B 0.000,C 180.000} C_DIS
LIN {X 106.536,Y 99.026,Z 80.070,A 180.000,B 0.000,C 180.000} C_DIS
LIN {X 106.560,Y 98.871,Z 80.066,A 180.000,B 0.000,C 180.000} C_DIS
LIN {X 106.583,Y 98.715,Z 80.062,A 180.000,B 0.000,C 180.000} C_DIS
LIN {X 106.605,Y 98.560,Z 80.059,A 180.000,B 0.000,C 180.000} C_DIS
LIN {X 106.625,Y 98.404,Z 80.056,A 180.000,B 0.000,C 180.000} C_DIS
LIN {X 106.640,Y 98.248,Z 80.052,A 180.000,B 0.000,C 180.000} C_DIS
LIN {X 106.654,Y 98.091,Z 80.049,A 180.000,B 0.000,C 180.000} C_DIS
LIN {X 106.664,Y 97.934,Z 80.046,A 180.000,B 0.000,C 180.000} C_DIS
LIN {X 106.670,Y 97.777,Z 80.043,A 180.000,B 0.000,C 180.000} C_DIS
LIN {X 106.675,Y 97.620,Z 80.040,A 180.000,B 0.000,C 180.000} C_DIS
LIN {X 106.677,Y 97.463,Z 80.037,A 180.000,B 0.000,C 180.000} C_DIS
LIN {X 106.676,Y 97.306,Z 80.035,A 180.000,B 0.000,C 180.000} C_DIS
LIN {X 106.673,Y 97.148,Z 80.032,A 180.000,B 0.000,C 180.000} C_DIS
LIN {X 106.658,Y 96.835,Z 80.027,A 180.000,B 0.000,C 180.000} C_DIS
LIN {X 106.632,Y 96.521,Z 80.022,A 180.000,B 0.000,C 180.000} C_DIS
LIN {X 106.593,Y 96.209,Z 80.018,A 180.000,B 0.000,C 180.000} C_DIS
LIN {X 106.549,Y 95.897,Z 80.014,A 180.000,B 0.000,C 180.000} C_DIS
LIN {X 106.489,Y 95.588,Z 80.011,A 180.000,B 0.000,C 180.000} C_DIS
LIN {X 106.417,Y 95.282,Z 80.008,A 180.000,B 0.000,C 180.000} C_DIS
LIN {X 106.339,Y 94.976,Z 80.006,A 180.000,B 0.000,C 180.000} C_DIS
LIN {X 106.248,Y 94.675,Z 80.003,A 180.000,B 0.000,C 180.000} C_DIS
LIN {X 106.147,Y 94.377,Z 80.002,A 180.000,B 0.000,C 180.000} C_DIS
LIN {X 106.034,Y 94.083,Z 80.001,A 180.000,B 0.000,C 180.000} C_DIS
LIN {X 105.914,Y 93.792,Z 80.000,A 180.000,B 0.000,C 180.000} C_DIS
LIN {X 105.810,Y 93.562,Z 80.000,A 180.000,B 0.000,C 180.000} C_DIS
; Cutting Move Starts
LIN {X 105.781,Y 93.500,Z 80.000,A 180.000,B 0.000,C 180.000} C_DIS
LIN {X 105.689,Y 93.321,Z 80.000,A 180.000,B 0.000,C 180.000} C_DIS
LIN {X 105.656,Y 93.257,Z 80.000,A 180.000,B 0.000,C 180.000} C_DIS
LIN {X 105.596,Y 93.142,Z 80.000,A 180.000,B 0.000,C 180.000} C_DIS
LIN {X 105.498,Y 92.964,Z 80.000,A 180.000,B 0.000,C 180.000} C_DIS
LIN {X 105.477,Y 92.928,Z 80.000,A 180.000,B 0.000,C 180.000} C_DIS
LIN {X 105.393,Y 92.785,Z 80.000,A 180.000,B 0.000,C 180.000} C_DIS
LIN {X 105.299,Y 92.626,Z 80.000,A 180.000,B 0.000,C 180.000} C_DIS
LIN {X 105.286,Y 92.606,Z 80.000,A 180.000,B 0.000,C 180.000} C_DIS
LIN {X 105.168,Y 92.427,Z 80.000,A 180.000,B 0.000,C 180.000} C_DIS
LIN {X 105.120,Y 92.355,Z 80.000,A 180.000,B 0.000,C 180.000} C_DIS
LIN {X 105.048,Y 92.249,Z 80.000,A 180.000,B 0.000,C 180.000} C_DIS
LIN {X 104.941,Y 92.101,Z 80.000,A 180.000,B 0.000,C 180.000} C_DIS
LIN {X 104.919,Y 92.070,Z 80.000,A 180.000,B 0.000,C 180.000} C_DIS
LIN {X 104.784,Y 91.891,Z 80.000,A 180.000,B 0.000,C 180.000} C_DIS
LIN {X 104.762,Y 91.862,Z 80.000,A 180.000,B 0.000,C 180.000} C_DIS
LIN {X 104.647,Y 91.712,Z 80.000,A 180.000,B 0.000,C 180.000} C_DIS
LIN {X 104.584,Y 91.637,Z 80.000,A 180.000,B 0.000,C 180.000} C_DIS
LIN {X 104.496,Y 91.533,Z 80.000,A 180.000,B 0.000,C 180.000} C_DIS
LIN {X 104.405,Y 91.426,Z 80.000,A 180.000,B 0.000,C 180.000} C_DIS
LIN {X 104.339,Y 91.355,Z 80.000,A 180.000,B 0.000,C 180.000} C_DIS
LIN {X 104.226,Y 91.234,Z 80.000,A 180.000,B 0.000,C 180.000} C_DIS
LIN {X 104.171,Y 91.176,Z 80.000,A 180.000,B 0.000,C 180.000} C_DIS
LIN {X 104.047,Y 91.045,Z 80.000,A 180.000,B 0.000,C 180.000} C_DIS
LIN {X 104.002,Y 90.997,Z 80.000,A 180.000,B 0.000,C 180.000} C_DIS
LIN {X 103.869,Y 90.868,Z 80.000,A 180.000,B 0.000,C 180.000} C_DIS
LIN {X 103.816,Y 90.818,Z 80.000,A 180.000,B 0.000,C 180.000} C_DIS
LIN {X 103.690,Y 90.699,Z 80.000,A 180.000,B 0.000,C 180.000} C_DIS
LIN {X 103.624,Y 90.640,Z 80.000,A 180.000,B 0.000,C 180.000} C_DIS
LIN {X 103.511,Y 90.544,Z 80.000,A 180.000,B 0.000,C 180.000} C_DIS
LIN {X 103.412,Y 90.461,Z 80.000,A 180.000,B 0.000,C 180.000} C_DIS
LIN {X 103.332,Y 90.394,Z 80.000,A 180.000,B 0.000,C 180.000} C_DIS
LIN {X 103.197,Y 90.282,Z 80.000,A 180.000,B 0.000,C 180.000} C_DIS
LIN {X 103.153,Y 90.248,Z 80.000,A 180.000,B 0.000,C 180.000} C_DIS
LIN {X 102.975,Y 90.113,Z 80.000,A 180.000,B 0.000,C 180.000} C_DIS
LIN {X 102.962,Y 90.103,Z 80.000,A 180.000,B 0.000,C 180.000} C_DIS
LIN {X 102.796,Y 89.982,Z 80.000,A 180.000,B 0.000,C 180.000} C_DIS
LIN {X 102.711,Y 89.925,Z 80.000,A 180.000,B 0.000,C 180.000} C_DIS
LIN {X 102.617,Y 89.862,Z 80.000,A 180.000,B 0.000,C 180.000} C_DIS
LIN {X 102.439,Y 89.746,Z 80.000,A 180.000,B 0.000,C 180.000} C_DIS
LIN {X 102.438,Y 89.745,Z 80.000,A 180.000,B 0.000,C 180.000} C_DIS
LIN {X 102.260,Y 89.633,Z 80.000,A 180.000,B 0.000,C 180.000} C_DIS
LIN {X 102.081,Y 89.528,Z 80.000,A 180.000,B 0.000,C 180.000} C_DIS
LIN {X 101.902,Y 89.426,Z 80.000,A 180.000,B 0.000,C 180.000} C_DIS
LIN {X 101.830,Y 89.388,Z 80.000,A 180.000,B 0.000,C 180.000} C_DIS
LIN {X 101.723,Y 89.333,Z 80.000,A 180.000,B 0.000,C 180.000} C_DIS
LIN {X 101.545,Y 89.243,Z 80.000,A 180.000,B 0.000,C 180.000} C_DIS
LIN {X 101.474,Y 89.209,Z 80.000,A 180.000,B 0.000,C 180.000} C_DIS
LIN {X 101.366,Y 89.158,Z 80.000,A 180.000,B 0.000,C 180.000} C_DIS
LIN {X 101.187,Y 89.078,Z 80.000,A 180.000,B 0.000,C 180.000} C_DIS
LIN {X 101.081,Y 89.031,Z 80.000,A 180.000,B 0.000,C 180.000} C_DIS
LIN {X 101.008,Y 88.999,Z 80.000,A 180.000,B 0.000,C 180.000} C_DIS
LIN {X 100.829,Y 88.929,Z 80.000,A 180.000,B 0.000,C 180.000} C_DIS
LIN {X 100.651,Y 88.861,Z 80.000,A 180.000,B 0.000,C 180.000} C_DIS
LIN {X 100.626,Y 88.852,Z 80.000,A 180.000,B 0.000,C 180.000} C_DIS
LIN {X 100.472,Y 88.800,Z 80.000,A 180.000,B 0.000,C 180.000} C_DIS
LIN {X 100.293,Y 88.742,Z 80.000,A 180.000,B 0.000,C 180.000} C_DIS
LIN {X 100.076,Y 88.673,Z 80.000,A 180.000,B 0.000,C 180.000} C_DIS
LIN {X 99.936,Y 88.633,Z 80.000,A 180.000,B 0.000,C 180.000} C_DIS
LIN {X 99.757,Y 88.586,Z 80.000,A 180.000,B 0.000,C 180.000} C_DIS
LIN {X 99.578,Y 88.542,Z 80.000,A 180.000,B 0.000,C 180.000} C_DIS
LIN {X 99.399,Y 88.505,Z 80.000,A 180.000,B 0.000,C 180.000} C_DIS
LIN {X 99.221,Y 88.470,Z 80.000,A 180.000,B 0.000,C 180.000} C_DIS
LIN {X 99.042,Y 88.436,Z 80.000,A 180.000,B 0.000,C 180.000} C_DIS
LIN {X 98.863,Y 88.407,Z 80.000,A 180.000,B 0.000,C 180.000} C_DIS
LIN {X 98.684,Y 88.381,Z 80.000,A 180.000,B 0.000,C 180.000} C_DIS
LIN {X 98.505,Y 88.359,Z 80.000,A 180.000,B 0.000,C 180.000} C_DIS
LIN {X 98.327,Y 88.344,Z 80.000,A 180.000,B 0.000,C 180.000} C_DIS
LIN {X 98.148,Y 88.329,Z 80.000,A 180.000,B 0.000,C 180.000} C_DIS
LIN {X 97.969,Y 88.318,Z 80.000,A 180.000,B 0.000,C 180.000} C_DIS
LIN {X 97.937,Y 88.316,Z 80.000,A 180.000,B 0.000,C 180.000} C_DIS
LIN {X 97.790,Y 88.310,Z 80.000,A 180.000,B 0.000,C 180.000} C_DIS
LIN {X 97.612,Y 88.305,Z 80.000,A 180.000,B 0.000,C 180.000} C_DIS
LIN {X 97.433,Y 88.304,Z 80.000,A 180.000,B 0.000,C 180.000} C_DIS
LIN {X 97.254,Y 88.309,Z 80.000,A 180.000,B 0.000,C 180.000} C_DIS
LIN {X 97.075,Y 88.315,Z 80.000,A 180.000,B 0.000,C 180.000} C_DIS
LIN {X 97.063,Y 88.316,Z 80.000,A 180.000,B 0.000,C 180.000} C_DIS
LIN {X 96.897,Y 88.326,Z 80.000,A 180.000,B 0.000,C 180.000} C_DIS
LIN {X 96.718,Y 88.340,Z 80.000,A 180.000,B 0.000,C 180.000} C_DIS
LIN {X 96.539,Y 88.355,Z 80.000,A 180.000,B 0.000,C 180.000} C_DIS
LIN {X 96.360,Y 88.375,Z 80.000,A 180.000,B 0.000,C 180.000} C_DIS
LIN {X 96.181,Y 88.400,Z 80.000,A 180.000,B 0.000,C 180.000} C_DIS
LIN {X 96.003,Y 88.427,Z 80.000,A 180.000,B 0.000,C 180.000} C_DIS
LIN {X 95.824,Y 88.461,Z 80.000,A 180.000,B 0.000,C 180.000} C_DIS
LIN {X 95.655,Y 88.494,Z 80.000,A 180.000,B 0.000,C 180.000} C_DIS
LIN {X 95.466,Y 88.532,Z 80.000,A 180.000,B 0.000,C 180.000} C_DIS
LIN {X 95.288,Y 88.575,Z 80.000,A 180.000,B 0.000,C 180.000} C_DIS
LIN {X 95.109,Y 88.621,Z 80.000,A 180.000,B 0.000,C 180.000} C_DIS
LIN {X 94.930,Y 88.671,Z 80.000,A 180.000,B 0.000,C 180.000} C_DIS
LIN {X 94.751,Y 88.728,Z 80.000,A 180.000,B 0.000,C 180.000} C_DIS
LIN {X 94.573,Y 88.786,Z 80.000,A 180.000,B 0.000,C 180.000} C_DIS
LIN {X 94.394,Y 88.845,Z 80.000,A 180.000,B 0.000,C 180.000} C_DIS
LIN {X 94.374,Y 88.852,Z 80.000,A 180.000,B 0.000,C 180.000} C_DIS
LIN {X 94.215,Y 88.912,Z 80.000,A 180.000,B 0.000,C 180.000} C_DIS
LIN {X 94.036,Y 88.981,Z 80.000,A 180.000,B 0.000,C 180.000} C_DIS
LIN {X 93.919,Y 89.031,Z 80.000,A 180.000,B 0.000,C 180.000} C_DIS
LIN {X 93.679,Y 89.138,Z 80.000,A 180.000,B 0.000,C 180.000} C_DIS
LIN {X 93.526,Y 89.209,Z 80.000,A 180.000,B 0.000,C 180.000} C_DIS
LIN {X 93.500,Y 89.222,Z 80.000,A 180.000,B 0.000,C 180.000} C_DIS
LIN {X 93.321,Y 89.310,Z 80.000,A 180.000,B 0.000,C 180.000} C_DIS
LIN {X 93.142,Y 89.403,Z 80.000,A 180.000,B 0.000,C 180.000} C_DIS
LIN {X 92.964,Y 89.502,Z 80.000,A 180.000,B 0.000,C 180.000} C_DIS
LIN {X 92.785,Y 89.607,Z 80.000,A 180.000,B 0.000,C 180.000} C_DIS
LIN {X 92.606,Y 89.717,Z 80.000,A 180.000,B 0.000,C 180.000} C_DIS
LIN {X 92.561,Y 89.746,Z 80.000,A 180.000,B 0.000,C 180.000} C_DIS
LIN {X 92.427,Y 89.832,Z 80.000,A 180.000,B 0.000,C 180.000} C_DIS
LIN {X 92.249,Y 89.952,Z 80.000,A 180.000,B 0.000,C 180.000} C_DIS
LIN {X 92.070,Y 90.079,Z 80.000,A 180.000,B 0.000,C 180.000} C_DIS
LIN {X 91.891,Y 90.214,Z 80.000,A 180.000,B 0.000,C 180.000} C_DIS
LIN {X 91.803,Y 90.282,Z 80.000,A 180.000,B 0.000,C 180.000} C_DIS
LIN {X 91.712,Y 90.357,Z 80.000,A 180.000,B 0.000,C 180.000} C_DIS
LIN {X 91.588,Y 90.461,Z 80.000,A 180.000,B 0.000,C 180.000} C_DIS
LIN {X 91.533,Y 90.507,Z 80.000,A 180.000,B 0.000,C 180.000} C_DIS
LIN {X 91.376,Y 90.640,Z 80.000,A 180.000,B 0.000,C 180.000} C_DIS
LIN {X 91.355,Y 90.658,Z 80.000,A 180.000,B 0.000,C 180.000} C_DIS
LIN {X 91.184,Y 90.818,Z 80.000,A 180.000,B 0.000,C 180.000} C_DIS
LIN {X 91.176,Y 90.826,Z 80.000,A 180.000,B 0.000,C 180.000} C_DIS
LIN {X 90.998,Y 90.997,Z 80.000,A 180.000,B 0.000,C 180.000} C_DIS
LIN {X 90.997,Y 90.998,Z 80.000,A 180.000,B 0.000,C 180.000} C_DIS
LIN {X 90.829,Y 91.176,Z 80.000,A 180.000,B 0.000,C 180.000} C_DIS
LIN {X 90.818,Y 91.187,Z 80.000,A 180.000,B 0.000,C 180.000} C_DIS
LIN {X 90.661,Y 91.355,Z 80.000,A 180.000,B 0.000,C 180.000} C_DIS
LIN {X 90.640,Y 91.377,Z 80.000,A 180.000,B 0.000,C 180.000} C_DIS
LIN {X 90.504,Y 91.533,Z 80.000,A 180.000,B 0.000,C 180.000} C_DIS
LIN {X 90.461,Y 91.585,Z 80.000,A 180.000,B 0.000,C 180.000} C_DIS
LIN {X 90.353,Y 91.712,Z 80.000,A 180.000,B 0.000,C 180.000} C_DIS
LIN {X 90.282,Y 91.803,Z 80.000,A 180.000,B 0.000,C 180.000} C_DIS
LIN {X 90.103,Y 92.040,Z 80.000,A 180.000,B 0.000,C 180.000} C_DIS
LIN {X 90.081,Y 92.070,Z 80.000,A 180.000,B 0.000,C 180.000} C_DIS
LIN {X 89.952,Y 92.249,Z 80.000,A 180.000,B 0.000,C 180.000} C_DIS
LIN {X 89.925,Y 92.288,Z 80.000,A 180.000,B 0.000,C 180.000} C_DIS
LIN {X 89.832,Y 92.427,Z 80.000,A 180.000,B 0.000,C 180.000} C_DIS
LIN {X 89.746,Y 92.556,Z 80.000,A 180.000,B 0.000,C 180.000} C_DIS
LIN {X 89.714,Y 92.606,Z 80.000,A 180.000,B 0.000,C 180.000} C_DIS
LIN {X 89.607,Y 92.785,Z 80.000,A 180.000,B 0.000,C 180.000} C_DIS
LIN {X 89.567,Y 92.853,Z 80.000,A 180.000,B 0.000,C 180.000} C_DIS
LIN {X 89.502,Y 92.964,Z 80.000,A 180.000,B 0.000,C 180.000} C_DIS
LIN {X 89.404,Y 93.142,Z 80.000,A 180.000,B 0.000,C 180.000} C_DIS
LIN {X 89.388,Y 93.172,Z 80.000,A 180.000,B 0.000,C 180.000} C_DIS
LIN {X 89.311,Y 93.321,Z 80.000,A 180.000,B 0.000,C 180.000} C_DIS
LIN {X 89.219,Y 93.500,Z 80.000,A 180.000,B 0.000,C 180.000} C_DIS
LIN {X 89.209,Y 93.519,Z 80.000,A 180.000,B 0.000,C 180.000} C_DIS
LIN {X 89.137,Y 93.679,Z 80.000,A 180.000,B 0.000,C 180.000} C_DIS
LIN {X 89.057,Y 93.857,Z 80.000,A 180.000,B 0.000,C 180.000} C_DIS
LIN {X 89.031,Y 93.919,Z 80.000,A 180.000,B 0.000,C 180.000} C_DIS
LIN {X 88.984,Y 94.036,Z 80.000,A 180.000,B 0.000,C 180.000} C_DIS
LIN {X 88.914,Y 94.215,Z 80.000,A 180.000,B 0.000,C 180.000} C_DIS
LIN {X 88.846,Y 94.394,Z 80.000,A 180.000,B 0.000,C 180.000} C_DIS
LIN {X 88.783,Y 94.573,Z 80.000,A 180.000,B 0.000,C 180.000} C_DIS
LIN {X 88.726,Y 94.751,Z 80.000,A 180.000,B 0.000,C 180.000} C_DIS
LIN {X 88.673,Y 94.921,Z 80.000,A 180.000,B 0.000,C 180.000} C_DIS
LIN {X 88.671,Y 94.930,Z 80.000,A 180.000,B 0.000,C 180.000} C_DIS
LIN {X 88.624,Y 95.109,Z 80.000,A 180.000,B 0.000,C 180.000} C_DIS
LIN {X 88.578,Y 95.288,Z 80.000,A 180.000,B 0.000,C 180.000} C_DIS
LIN {X 88.532,Y 95.466,Z 80.000,A 180.000,B 0.000,C 180.000} C_DIS
LIN {X 88.494,Y 95.644,Z 80.000,A 180.000,B 0.000,C 180.000} C_DIS
LIN {X 88.459,Y 95.824,Z 80.000,A 180.000,B 0.000,C 180.000} C_DIS
LIN {X 88.427,Y 96.003,Z 80.000,A 180.000,B 0.000,C 180.000} C_DIS
LIN {X 88.402,Y 96.181,Z 80.000,A 180.000,B 0.000,C 180.000} C_DIS
LIN {X 88.377,Y 96.360,Z 80.000,A 180.000,B 0.000,C 180.000} C_DIS
LIN {X 88.366,Y 96.452,Z 80.000,A 180.000,B 0.000,C 180.000} C_DIS
LIN {X 88.355,Y 96.539,Z 80.000,A 180.000,B 0.000,C 180.000} C_DIS
LIN {X 88.339,Y 96.718,Z 80.000,A 180.000,B 0.000,C 180.000} C_DIS
LIN {X 88.324,Y 96.897,Z 80.000,A 180.000,B 0.000,C 180.000} C_DIS
LIN {X 88.316,Y 97.036,Z 80.000,A 180.000,B 0.000,C 180.000} C_DIS
LIN {X 88.314,Y 97.075,Z 80.000,A 180.000,B 0.000,C 180.000} C_DIS
LIN {X 88.309,Y 97.254,Z 80.000,A 180.000,B 0.000,C 180.000} C_DIS
LIN {X 88.306,Y 97.433,Z 80.000,A 180.000,B 0.000,C 180.000} C_DIS
LIN {X 88.306,Y 97.612,Z 80.000,A 180.000,B 0.000,C 180.000} C_DIS
LIN {X 88.311,Y 97.790,Z 80.000,A 180.000,B 0.000,C 180.000} C_DIS
LIN {X 88.316,Y 97.964,Z 80.000,A 180.000,B 0.000,C 180.000} C_DIS
LIN {X 88.316,Y 97.969,Z 80.000,A 180.000,B 0.000,C 180.000} C_DIS
LIN {X 88.328,Y 98.148,Z 80.000,A 180.000,B 0.000,C 180.000} C_DIS
LIN {X 88.343,Y 98.327,Z 80.000,A 180.000,B 0.000,C 180.000} C_DIS
LIN {X 88.361,Y 98.505,Z 80.000,A 180.000,B 0.000,C 180.000} C_DIS
LIN {X 88.383,Y 98.684,Z 80.000,A 180.000,B 0.000,C 180.000} C_DIS
LIN {X 88.408,Y 98.863,Z 80.000,A 180.000,B 0.000,C 180.000} C_DIS
LIN {X 88.434,Y 99.042,Z 80.000,A 180.000,B 0.000,C 180.000} C_DIS
LIN {X 88.467,Y 99.221,Z 80.000,A 180.000,B 0.000,C 180.000} C_DIS
LIN {X 88.503,Y 99.399,Z 80.000,A 180.000,B 0.000,C 180.000} C_DIS
LIN {X 88.543,Y 99.578,Z 80.000,A 180.000,B 0.000,C 180.000} C_DIS
LIN {X 88.589,Y 99.757,Z 80.000,A 180.000,B 0.000,C 180.000} C_DIS
LIN {X 88.635,Y 99.936,Z 80.000,A 180.000,B 0.000,C 180.000} C_DIS
LIN {X 88.673,Y 100.079,Z 80.000,A 180.000,B 0.000,C 180.000} C_DIS
LIN {X 88.683,Y 100.114,Z 80.000,A 180.000,B 0.000,C 180.000} C_DIS
LIN {X 88.740,Y 100.293,Z 80.000,A 180.000,B 0.000,C 180.000} C_DIS
LIN {X 88.797,Y 100.472,Z 80.000,A 180.000,B 0.000,C 180.000} C_DIS
LIN {X 88.852,Y 100.622,Z 80.000,A 180.000,B 0.000,C 180.000} C_DIS
LIN {X 88.931,Y 100.829,Z 80.000,A 180.000,B 0.000,C 180.000} C_DIS
LIN {X 89.001,Y 101.008,Z 80.000,A 180.000,B 0.000,C 180.000} C_DIS
LIN {X 89.031,Y 101.081,Z 80.000,A 180.000,B 0.000,C 180.000} C_DIS
LIN {X 89.077,Y 101.187,Z 80.000,A 180.000,B 0.000,C 180.000} C_DIS
LIN {X 89.157,Y 101.366,Z 80.000,A 180.000,B 0.000,C 180.000} C_DIS
LIN {X 89.209,Y 101.481,Z 80.000,A 180.000,B 0.000,C 180.000} C_DIS
LIN {X 89.241,Y 101.545,Z 80.000,A 180.000,B 0.000,C 180.000} C_DIS
LIN {X 89.334,Y 101.723,Z 80.000,A 180.000,B 0.000,C 180.000} C_DIS
LIN {X 89.388,Y 101.828,Z 80.000,A 180.000,B 0.000,C 180.000} C_DIS
LIN {X 89.428,Y 101.902,Z 80.000,A 180.000,B 0.000,C 180.000} C_DIS
LIN {X 89.528,Y 102.081,Z 80.000,A 180.000,B 0.000,C 180.000} C_DIS
LIN {X 89.633,Y 102.260,Z 80.000,A 180.000,B 0.000,C 180.000} C_DIS
LIN {X 89.742,Y 102.438,Z 80.000,A 180.000,B 0.000,C 180.000} C_DIS
LIN {X 89.746,Y 102.444,Z 80.000,A 180.000,B 0.000,C 180.000} C_DIS
LIN {X 89.861,Y 102.617,Z 80.000,A 180.000,B 0.000,C 180.000} C_DIS
LIN {X 89.925,Y 102.712,Z 80.000,A 180.000,B 0.000,C 180.000} C_DIS
LIN {X 89.984,Y 102.796,Z 80.000,A 180.000,B 0.000,C 180.000} C_DIS
LIN {X 90.103,Y 102.960,Z 80.000,A 180.000,B 0.000,C 180.000} C_DIS
LIN {X 90.282,Y 103.197,Z 80.000,A 180.000,B 0.000,C 180.000} C_DIS
LIN {X 90.391,Y 103.332,Z 80.000,A 180.000,B 0.000,C 180.000} C_DIS
LIN {X 90.542,Y 103.511,Z 80.000,A 180.000,B 0.000,C 180.000} C_DIS
LIN {X 90.640,Y 103.623,Z 80.000,A 180.000,B 0.000,C 180.000} C_DIS
LIN {X 90.703,Y 103.690,Z 80.000,A 180.000,B 0.000,C 180.000} C_DIS
LIN {X 90.818,Y 103.813,Z 80.000,A 180.000,B 0.000,C 180.000} C_DIS
LIN {X 90.871,Y 103.869,Z 80.000,A 180.000,B 0.000,C 180.000} C_DIS
LIN {X 90.997,Y 104.002,Z 80.000,A 180.000,B 0.000,C 180.000} C_DIS
LIN {X 91.042,Y 104.047,Z 80.000,A 180.000,B 0.000,C 180.000} C_DIS
LIN {X 91.176,Y 104.174,Z 80.000,A 180.000,B 0.000,C 180.000} C_DIS
LIN {X 91.231,Y 104.226,Z 80.000,A 180.000,B 0.000,C 180.000} C_DIS
LIN {X 91.355,Y 104.342,Z 80.000,A 180.000,B 0.000,C 180.000} C_DIS
LIN {X 91.429,Y 104.405,Z 80.000,A 180.000,B 0.000,C 180.000} C_DIS
LIN {X 91.533,Y 104.493,Z 80.000,A 180.000,B 0.000,C 180.000} C_DIS
LIN {X 91.640,Y 104.584,Z 80.000,A 180.000,B 0.000,C 180.000} C_DIS
LIN {X 91.712,Y 104.643,Z 80.000,A 180.000,B 0.000,C 180.000} C_DIS
LIN {X 91.860,Y 104.762,Z 80.000,A 180.000,B 0.000,C 180.000} C_DIS
LIN {X 91.891,Y 104.786,Z 80.000,A 180.000,B 0.000,C 180.000} C_DIS
LIN {X 92.097,Y 104.941,Z 80.000,A 180.000,B 0.000,C 180.000} C_DIS
LIN {X 92.249,Y 105.048,Z 80.000,A 180.000,B 0.000,C 180.000} C_DIS
LIN {X 92.427,Y 105.168,Z 80.000,A 180.000,B 0.000,C 180.000} C_DIS
LIN {X 92.606,Y 105.283,Z 80.000,A 180.000,B 0.000,C 180.000} C_DIS
LIN {X 92.631,Y 105.299,Z 80.000,A 180.000,B 0.000,C 180.000} C_DIS
LIN {X 92.785,Y 105.393,Z 80.000,A 180.000,B 0.000,C 180.000} C_DIS
LIN {X 92.964,Y 105.498,Z 80.000,A 180.000,B 0.000,C 180.000} C_DIS
LIN {X 93.142,Y 105.597,Z 80.000,A 180.000,B 0.000,C 180.000} C_DIS
LIN {X 93.321,Y 105.690,Z 80.000,A 180.000,B 0.000,C 180.000} C_DIS
LIN {X 93.500,Y 105.778,Z 80.000,A 180.000,B 0.000,C 180.000} C_DIS
LIN {X 93.620,Y 105.835,Z 80.000,A 180.000,B 0.000,C 180.000} C_DIS
LIN {X 93.679,Y 105.862,Z 80.000,A 180.000,B 0.000,C 180.000} C_DIS
LIN {X 93.857,Y 105.942,Z 80.000,A 180.000,B 0.000,C 180.000} C_DIS
LIN {X 94.023,Y 106.014,Z 80.000,A 180.000,B 0.000,C 180.000} C_DIS
LIN {X 94.036,Y 106.019,Z 80.000,A 180.000,B 0.000,C 180.000} C_DIS
LIN {X 94.215,Y 106.088,Z 80.000,A 180.000,B 0.000,C 180.000} C_DIS
LIN {X 94.394,Y 106.155,Z 80.000,A 180.000,B 0.000,C 180.000} C_DIS
LIN {X 94.505,Y 106.193,Z 80.000,A 180.000,B 0.000,C 180.000} C_DIS
LIN {X 94.573,Y 106.214,Z 80.000,A 180.000,B 0.000,C 180.000} C_DIS
LIN {X 94.751,Y 106.272,Z 80.000,A 180.000,B 0.000,C 180.000} C_DIS
LIN {X 94.930,Y 106.329,Z 80.000,A 180.000,B 0.000,C 180.000} C_DIS
LIN {X 95.080,Y 106.371,Z 80.000,A 180.000,B 0.000,C 180.000} C_DIS
LIN {X 95.288,Y 106.425,Z 80.000,A 180.000,B 0.000,C 180.000} C_DIS
LIN {X 95.466,Y 106.468,Z 80.000,A 180.000,B 0.000,C 180.000} C_DIS
LIN {X 95.645,Y 106.504,Z 80.000,A 180.000,B 0.000,C 180.000} C_DIS
LIN {X 95.824,Y 106.539,Z 80.000,A 180.000,B 0.000,C 180.000} C_DIS
LIN {X 95.883,Y 106.550,Z 80.000,A 180.000,B 0.000,C 180.000} C_DIS
LIN {X 96.003,Y 106.573,Z 80.000,A 180.000,B 0.000,C 180.000} C_DIS
LIN {X 96.181,Y 106.600,Z 80.000,A 180.000,B 0.000,C 180.000} C_DIS
LIN {X 96.360,Y 106.625,Z 80.000,A 180.000,B 0.000,C 180.000} C_DIS
LIN {X 96.539,Y 106.645,Z 80.000,A 180.000,B 0.000,C 180.000} C_DIS
LIN {X 96.718,Y 106.660,Z 80.000,A 180.000,B 0.000,C 180.000} C_DIS
LIN {X 96.897,Y 106.674,Z 80.000,A 180.000,B 0.000,C 180.000} C_DIS
LIN {X 97.075,Y 106.685,Z 80.000,A 180.000,B 0.000,C 180.000} C_DIS
LIN {X 97.254,Y 106.691,Z 80.000,A 180.000,B 0.000,C 180.000} C_DIS
LIN {X 97.433,Y 106.696,Z 80.000,A 180.000,B 0.000,C 180.000} C_DIS
LIN {X 97.612,Y 106.695,Z 80.000,A 180.000,B 0.000,C 180.000} C_DIS
LIN {X 97.790,Y 106.690,Z 80.000,A 180.000,B 0.000,C 180.000} C_DIS
LIN {X 97.969,Y 106.682,Z 80.000,A 180.000,B 0.000,C 180.000} C_DIS
LIN {X 98.148,Y 106.671,Z 80.000,A 180.000,B 0.000,C 180.000} C_DIS
LIN {X 98.327,Y 106.656,Z 80.000,A 180.000,B 0.000,C 180.000} C_DIS
LIN {X 98.505,Y 106.641,Z 80.000,A 180.000,B 0.000,C 180.000} C_DIS
LIN {X 98.684,Y 106.619,Z 80.000,A 180.000,B 0.000,C 180.000} C_DIS
LIN {X 98.863,Y 106.593,Z 80.000,A 180.000,B 0.000,C 180.000} C_DIS
LIN {X 99.042,Y 106.564,Z 80.000,A 180.000,B 0.000,C 180.000} C_DIS
LIN {X 99.117,Y 106.550,Z 80.000,A 180.000,B 0.000,C 180.000} C_DIS
LIN {X 99.221,Y 106.530,Z 80.000,A 180.000,B 0.000,C 180.000} C_DIS
LIN {X 99.399,Y 106.495,Z 80.000,A 180.000,B 0.000,C 180.000} C_DIS
LIN {X 99.578,Y 106.458,Z 80.000,A 180.000,B 0.000,C 180.000} C_DIS
LIN {X 99.757,Y 106.414,Z 80.000,A 180.000,B 0.000,C 180.000} C_DIS
LIN {X 99.936,Y 106.367,Z 80.000,A 180.000,B 0.000,C 180.000} C_DIS
LIN {X 100.114,Y 106.315,Z 80.000,A 180.000,B 0.000,C 180.000} C_DIS
LIN {X 100.293,Y 106.258,Z 80.000,A 180.000,B 0.000,C 180.000} C_DIS
LIN {X 100.472,Y 106.200,Z 80.000,A 180.000,B 0.000,C 180.000} C_DIS
LIN {X 100.495,Y 106.193,Z 80.000,A 180.000,B 0.000,C 180.000} C_DIS
LIN {X 100.651,Y 106.139,Z 80.000,A 180.000,B 0.000,C 180.000} C_DIS
LIN {X 100.829,Y 106.071,Z 80.000,A 180.000,B 0.000,C 180.000} C_DIS
LIN {X 100.977,Y 106.014,Z 80.000,A 180.000,B 0.000,C 180.000} C_DIS
LIN {X 101.008,Y 106.001,Z 80.000,A 180.000,B 0.000,C 180.000} C_DIS
LIN {X 101.187,Y 105.922,Z 80.000,A 180.000,B 0.000,C 180.000} C_DIS
LIN {X 101.366,Y 105.842,Z 80.000,A 180.000,B 0.000,C 180.000} C_DIS
LIN {X 101.380,Y 105.835,Z 80.000,A 180.000,B 0.000,C 180.000} C_DIS
LIN {X 101.545,Y 105.757,Z 80.000,A 180.000,B 0.000,C 180.000} C_DIS
LIN {X 101.723,Y 105.667,Z 80.000,A 180.000,B 0.000,C 180.000} C_DIS
LIN {X 101.744,Y 105.656,Z 80.000,A 180.000,B 0.000,C 180.000} C_DIS
LIN {X 101.902,Y 105.574,Z 80.000,A 180.000,B 0.000,C 180.000} C_DIS
LIN {X 102.072,Y 105.477,Z 80.000,A 180.000,B 0.000,C 180.000} C_DIS
LIN {X 102.260,Y 105.367,Z 80.000,A 180.000,B 0.000,C 180.000} C_DIS
LIN {X 102.369,Y 105.299,Z 80.000,A 180.000,B 0.000,C 180.000} C_DIS
LIN {X 102.438,Y 105.255,Z 80.000,A 180.000,B 0.000,C 180.000} C_DIS
LIN {X 102.617,Y 105.138,Z 80.000,A 180.000,B 0.000,C 180.000} C_DIS
LIN {X 102.644,Y 105.120,Z 80.000,A 180.000,B 0.000,C 180.000} C_DIS
LIN {X 102.796,Y 105.018,Z 80.000,A 180.000,B 0.000,C 180.000} C_DIS
LIN {X 102.903,Y 104.941,Z 80.000,A 180.000,B 0.000,C 180.000} C_DIS
LIN {X 102.975,Y 104.887,Z 80.000,A 180.000,B 0.000,C 180.000} C_DIS
LIN {X 103.140,Y 104.762,Z 80.000,A 180.000,B 0.000,C 180.000} C_DIS
LIN {X 103.153,Y 104.752,Z 80.000,A 180.000,B 0.000,C 180.000} C_DIS
LIN {X 103.332,Y 104.606,Z 80.000,A 180.000,B 0.000,C 180.000} C_DIS
LIN {X 103.360,Y 104.584,Z 80.000,A 180.000,B 0.000,C 180.000} C_DIS
LIN {X 103.511,Y 104.456,Z 80.000,A 180.000,B 0.000,C 180.000} C_DIS
LIN {X 103.571,Y 104.405,Z 80.000,A 180.000,B 0.000,C 180.000} C_DIS
LIN {X 103.690,Y 104.301,Z 80.000,A 180.000,B 0.000,C 180.000} C_DIS
LIN {X 103.769,Y 104.226,Z 80.000,A 180.000,B 0.000,C 180.000} C_DIS
LIN {X 103.869,Y 104.132,Z 80.000,A 180.000,B 0.000,C 180.000} C_DIS
LIN {X 103.958,Y 104.047,Z 80.000,A 180.000,B 0.000,C 180.000} C_DIS
LIN {X 104.047,Y 103.955,Z 80.000,A 180.000,B 0.000,C 180.000} C_DIS
LIN {X 104.226,Y 103.766,Z 80.000,A 180.000,B 0.000,C 180.000} C_DIS
LIN {X 104.297,Y 103.690,Z 80.000,A 180.000,B 0.000,C 180.000} C_DIS
LIN {X 104.405,Y 103.574,Z 80.000,A 180.000,B 0.000,C 180.000} C_DIS
LIN {X 104.458,Y 103.511,Z 80.000,A 180.000,B 0.000,C 180.000} C_DIS
LIN {X 104.609,Y 103.332,Z 80.000,A 180.000,B 0.000,C 180.000} C_DIS
LIN {X 104.751,Y 103.153,Z 80.000,A 180.000,B 0.000,C 180.000} C_DIS
LIN {X 104.886,Y 102.975,Z 80.000,A 180.000,B 0.000,C 180.000} C_DIS
LIN {X 104.941,Y 102.899,Z 80.000,A 180.000,B 0.000,C 180.000} C_DIS
LIN {X 105.016,Y 102.796,Z 80.000,A 180.000,B 0.000,C 180.000} C_DIS
LIN {X 105.120,Y 102.645,Z 80.000,A 180.000,B 0.000,C 180.000} C_DIS
LIN {X 105.139,Y 102.617,Z 80.000,A 180.000,B 0.000,C 180.000} C_DIS
LIN {X 105.258,Y 102.438,Z 80.000,A 180.000,B 0.000,C 180.000} C_DIS
LIN {X 105.299,Y 102.374,Z 80.000,A 180.000,B 0.000,C 180.000} C_DIS
LIN {X 105.367,Y 102.260,Z 80.000,A 180.000,B 0.000,C 180.000} C_DIS
LIN {X 105.472,Y 102.081,Z 80.000,A 180.000,B 0.000,C 180.000} C_DIS
LIN {X 105.477,Y 102.072,Z 80.000,A 180.000,B 0.000,C 180.000} C_DIS
LIN {X 105.572,Y 101.902,Z 80.000,A 180.000,B 0.000,C 180.000} C_DIS
LIN {X 105.656,Y 101.743,Z 80.000,A 180.000,B 0.000,C 180.000} C_DIS
LIN {X 105.759,Y 101.545,Z 80.000,A 180.000,B 0.000,C 180.000} C_DIS
LIN {X 105.835,Y 101.384,Z 80.000,A 180.000,B 0.000,C 180.000} C_DIS
LIN {X 105.923,Y 101.187,Z 80.000,A 180.000,B 0.000,C 180.000} C_DIS
LIN {X 105.999,Y 101.008,Z 80.000,A 180.000,B 0.000,C 180.000} C_DIS
LIN {X 106.014,Y 100.970,Z 80.000,A 180.000,B 0.000,C 180.000} C_DIS
LIN {X 106.069,Y 100.829,Z 80.000,A 180.000,B 0.000,C 180.000} C_DIS
LIN {X 106.137,Y 100.651,Z 80.000,A 180.000,B 0.000,C 180.000} C_DIS
LIN {X 106.193,Y 100.502,Z 80.000,A 180.000,B 0.000,C 180.000} C_DIS
LIN {X 106.203,Y 100.472,Z 80.000,A 180.000,B 0.000,C 180.000} C_DIS
LIN {X 106.260,Y 100.293,Z 80.000,A 180.000,B 0.000,C 180.000} C_DIS
LIN {X 106.317,Y 100.114,Z 80.000,A 180.000,B 0.000,C 180.000} C_DIS
LIN {X 106.365,Y 99.936,Z 80.000,A 180.000,B 0.000,C 180.000} C_DIS
LIN {X 106.411,Y 99.757,Z 80.000,A 180.000,B 0.000,C 180.000} C_DIS
LIN {X 106.457,Y 99.578,Z 80.000,A 180.000,B 0.000,C 180.000} C_DIS
LIN {X 106.497,Y 99.399,Z 80.000,A 180.000,B 0.000,C 180.000} C_DIS
LIN {X 106.533,Y 99.221,Z 80.000,A 180.000,B 0.000,C 180.000} C_DIS
LIN {X 106.550,Y 99.132,Z 80.000,A 180.000,B 0.000,C 180.000} C_DIS
LIN {X 106.566,Y 99.042,Z 80.000,A 180.000,B 0.000,C 180.000} C_DIS
LIN {X 106.592,Y 98.863,Z 80.000,A 180.000,B 0.000,C 180.000} C_DIS
LIN {X 106.617,Y 98.684,Z 80.000,A 180.000,B 0.000,C 180.000} C_DIS
LIN {X 106.639,Y 98.505,Z 80.000,A 180.000,B 0.000,C 180.000} C_DIS
LIN {X 106.657,Y 98.327,Z 80.000,A 180.000,B 0.000,C 180.000} C_DIS
LIN {X 106.672,Y 98.148,Z 80.000,A 180.000,B 0.000,C 180.000} C_DIS
LIN {X 106.684,Y 97.969,Z 80.000,A 180.000,B 0.000,C 180.000} C_DIS
LIN {X 106.689,Y 97.790,Z 80.000,A 180.000,B 0.000,C 180.000} C_DIS
LIN {X 106.694,Y 97.612,Z 80.000,A 180.000,B 0.000,C 180.000} C_DIS
LIN {X 106.694,Y 97.433,Z 80.000,A 180.000,B 0.000,C 180.000} C_DIS
LIN {X 106.691,Y 97.254,Z 80.000,A 180.000,B 0.000,C 180.000} C_DIS
LIN {X 106.686,Y 97.075,Z 80.000,A 180.000,B 0.000,C 180.000} C_DIS
LIN {X 106.676,Y 96.897,Z 80.000,A 180.000,B 0.000,C 180.000} C_DIS
LIN {X 106.661,Y 96.718,Z 80.000,A 180.000,B 0.000,C 180.000} C_DIS
LIN {X 106.645,Y 96.539,Z 80.000,A 180.000,B 0.000,C 180.000} C_DIS
LIN {X 106.623,Y 96.360,Z 80.000,A 180.000,B 0.000,C 180.000} C_DIS
LIN {X 106.598,Y 96.181,Z 80.000,A 180.000,B 0.000,C 180.000} C_DIS
LIN {X 106.573,Y 96.003,Z 80.000,A 180.000,B 0.000,C 180.000} C_DIS
LIN {X 106.550,Y 95.868,Z 80.000,A 180.000,B 0.000,C 180.000} C_DIS
LIN {X 106.541,Y 95.824,Z 80.000,A 180.000,B 0.000,C 180.000} C_DIS
LIN {X 106.506,Y 95.645,Z 80.000,A 180.000,B 0.000,C 180.000} C_DIS
LIN {X 106.468,Y 95.466,Z 80.000,A 180.000,B 0.000,C 180.000} C_DIS
LIN {X 106.422,Y 95.288,Z 80.000,A 180.000,B 0.000,C 180.000} C_DIS
LIN {X 106.371,Y 95.091,Z 80.000,A 180.000,B 0.000,C 180.000} C_DIS
LIN {X 106.329,Y 94.930,Z 80.000,A 180.000,B 0.000,C 180.000} C_DIS
LIN {X 106.274,Y 94.751,Z 80.000,A 180.000,B 0.000,C 180.000} C_DIS
LIN {X 106.217,Y 94.573,Z 80.000,A 180.000,B 0.000,C 180.000} C_DIS
LIN {X 106.193,Y 94.498,Z 80.000,A 180.000,B 0.000,C 180.000} C_DIS
LIN {X 106.154,Y 94.394,Z 80.000,A 180.000,B 0.000,C 180.000} C_DIS
LIN {X 106.086,Y 94.215,Z 80.000,A 180.000,B 0.000,C 180.000} C_DIS
LIN {X 106.016,Y 94.036,Z 80.000,A 180.000,B 0.000,C 180.000} C_DIS
LIN {X 106.014,Y 94.030,Z 80.000,A 180.000,B 0.000,C 180.000} C_DIS
LIN {X 105.943,Y 93.857,Z 80.000,A 180.000,B 0.000,C 180.000} C_DIS
LIN {X 105.835,Y 93.616,Z 80.000,A 180.000,B 0.000,C 180.000} C_DIS
LIN {X 105.810,Y 93.562,Z 80.000,A 180.000,B 0.000,C 180.000} C_DIS
; Link Move Starts
LIN {X 105.679,Y 93.302,Z 80.000,A 180.000,B 0.000,C 180.000} C_DIS
LIN {X 105.537,Y 93.034,Z 79.999,A 180.000,B 0.000,C 180.000} C_DIS
LIN {X 105.387,Y 92.773,Z 79.998,A 180.000,B 0.000,C 180.000} C_DIS
LIN {X 105.236,Y 92.526,Z 79.997,A 180.000,B 0.000,C 180.000} C_DIS
LIN {X 105.068,Y 92.273,Z 79.995,A 180.000,B 0.000,C 180.000} C_DIS
LIN {X 104.893,Y 92.029,Z 79.992,A 180.000,B 0.000,C 180.000} C_DIS
LIN {X 104.714,Y 91.789,Z 79.990,A 180.000,B 0.000,C 180.000} C_DIS
LIN {X 104.522,Y 91.554,Z 79.986,A 180.000,B 0.000,C 180.000} C_DIS
LIN {X 104.328,Y 91.331,Z 79.983,A 180.000,B 0.000,C 180.000} C_DIS
LIN {X 104.117,Y 91.105,Z 79.979,A 180.000,B 0.000,C 180.000} C_DIS
LIN {X 103.913,Y 90.894,Z 79.975,A 180.000,B 0.000,C 180.000} C_DIS
LIN {X 103.695,Y 90.684,Z 79.970,A 180.000,B 0.000,C 180.000} C_DIS
LIN {X 103.470,Y 90.488,Z 79.965,A 180.000,B 0.000,C 180.000} C_DIS
LIN {X 103.352,Y 90.387,Z 79.962,A 180.000,B 0.000,C 180.000} C_DIS
LIN {X 103.233,Y 90.287,Z 79.959,A 180.000,B 0.000,C 180.000} C_DIS
LIN {X 103.118,Y 90.195,Z 79.957,A 180.000,B 0.000,C 180.000} C_DIS
LIN {X 103.002,Y 90.106,Z 79.954,A 180.000,B 0.000,C 180.000} C_DIS
LIN {X 102.885,Y 90.017,Z 79.951,A 180.000,B 0.000,C 180.000} C_DIS
LIN {X 102.765,Y 89.932,Z 79.948,A 180.000,B 0.000,C 180.000} C_DIS
LIN {X 102.637,Y 89.845,Z 79.944,A 180.000,B 0.000,C 180.000} C_DIS
LIN {X 102.509,Y 89.758,Z 79.941,A 180.000,B 0.000,C 180.000} C_DIS
LIN {X 102.384,Y 89.676,Z 79.938,A 180.000,B 0.000,C 180.000} C_DIS
LIN {X 102.258,Y 89.597,Z 79.934,A 180.000,B 0.000,C 180.000} C_DIS
LIN {X 102.128,Y 89.518,Z 79.931,A 180.000,B 0.000,C 180.000} C_DIS
LIN {X 101.999,Y 89.440,Z 79.927,A 180.000,B 0.000,C 180.000} C_DIS
LIN {X 101.869,Y 89.368,Z 79.924,A 180.000,B 0.000,C 180.000} C_DIS
LIN {X 101.738,Y 89.299,Z 79.920,A 180.000,B 0.000,C 180.000} C_DIS
LIN {X 101.606,Y 89.229,Z 79.916,A 180.000,B 0.000,C 180.000} C_DIS
LIN {X 101.472,Y 89.163,Z 79.913,A 180.000,B 0.000,C 180.000} C_DIS
LIN {X 101.334,Y 89.097,Z 79.908,A 180.000,B 0.000,C 180.000} C_DIS
LIN {X 101.194,Y 89.033,Z 79.904,A 180.000,B 0.000,C 180.000} C_DIS
LIN {X 101.060,Y 88.971,Z 79.900,A 180.000,B 0.000,C 180.000} C_DIS
LIN {X 100.924,Y 88.914,Z 79.896,A 180.000,B 0.000,C 180.000} C_DIS
LIN {X 100.785,Y 88.858,Z 79.892,A 180.000,B 0.000,C 180.000} C_DIS
LIN {X 100.645,Y 88.803,Z 79.888,A 180.000,B 0.000,C 180.000} C_DIS
LIN {X 100.502,Y 88.752,Z 79.883,A 180.000,B 0.000,C 180.000} C_DIS
LIN {X 100.358,Y 88.704,Z 79.879,A 180.000,B 0.000,C 180.000} C_DIS
LIN {X 100.210,Y 88.654,Z 79.874,A 180.000,B 0.000,C 180.000} C_DIS
LIN {X 100.063,Y 88.605,Z 79.870,A 180.000,B 0.000,C 180.000} C_DIS
LIN {X 99.921,Y 88.564,Z 79.865,A 180.000,B 0.000,C 180.000} C_DIS
LIN {X 99.778,Y 88.525,Z 79.861,A 180.000,B 0.000,C 180.000} C_DIS
LIN {X 99.637,Y 88.486,Z 79.856,A 180.000,B 0.000,C 180.000} C_DIS
LIN {X 99.494,Y 88.453,Z 79.851,A 180.000,B 0.000,C 180.000} C_DIS
LIN {X 99.417,Y 88.437,Z 79.849,A 180.000,B 0.000,C 180.000} C_DIS
LIN {X 99.341,Y 88.420,Z 79.846,A 180.000,B 0.000,C 180.000} C_DIS
LIN {X 99.264,Y 88.404,Z 79.844,A 180.000,B 0.000,C 180.000} C_DIS
LIN {X 99.187,Y 88.388,Z 79.841,A 180.000,B 0.000,C 180.000} C_DIS
LIN {X 99.043,Y 88.358,Z 79.836,A 180.000,B 0.000,C 180.000} C_DIS
LIN {X 98.898,Y 88.332,Z 79.831,A 180.000,B 0.000,C 180.000} C_DIS
LIN {X 98.823,Y 88.320,Z 79.829,A 180.000,B 0.000,C 180.000} C_DIS
LIN {X 98.673,Y 88.297,Z 79.824,A 180.000,B 0.000,C 180.000} C_DIS
LIN {X 98.598,Y 88.285,Z 79.821,A 180.000,B 0.000,C 180.000} C_DIS
LIN {X 98.523,Y 88.275,Z 79.818,A 180.000,B 0.000,C 180.000} C_DIS
LIN {X 98.447,Y 88.268,Z 79.816,A 180.000,B 0.000,C 180.000} C_DIS
LIN {X 98.219,Y 88.245,Z 79.808,A 180.000,B 0.000,C 180.000} C_DIS
LIN {X 98.143,Y 88.237,Z 79.805,A 180.000,B 0.000,C 180.000} C_DIS
LIN {X 97.989,Y 88.225,Z 79.800,A 180.000,B 0.000,C 180.000} C_DIS
LIN {X 97.914,Y 88.220,Z 79.797,A 180.000,B 0.000,C 180.000} C_DIS
LIN {X 97.838,Y 88.216,Z 79.795,A 180.000,B 0.000,C 180.000} C_DIS
LIN {X 97.614,Y 88.206,Z 79.787,A 180.000,B 0.000,C 180.000} C_DIS
LIN {X 97.540,Y 88.203,Z 79.784,A 180.000,B 0.000,C 180.000} C_DIS
LIN {X 97.467,Y 88.202,Z 79.782,A 180.000,B 0.000,C 180.000} C_DIS
LIN {X 97.393,Y 88.202,Z 79.779,A 180.000,B 0.000,C 180.000} C_DIS
LIN {X 97.241,Y 88.204,Z 79.774,A 180.000,B 0.000,C 180.000} C_DIS
LIN {X 97.165,Y 88.205,Z 79.771,A 180.000,B 0.000,C 180.000} C_DIS
LIN {X 97.089,Y 88.206,Z 79.768,A 180.000,B 0.000,C 180.000} C_DIS
LIN {X 97.012,Y 88.209,Z 79.766,A 180.000,B 0.000,C 180.000} C_DIS
LIN {X 96.857,Y 88.216,Z 79.760,A 180.000,B 0.000,C 180.000} C_DIS
LIN {X 96.780,Y 88.221,Z 79.758,A 180.000,B 0.000,C 180.000} C_DIS
LIN {X 96.627,Y 88.232,Z 79.752,A 180.000,B 0.000,C 180.000} C_DIS
LIN {X 96.550,Y 88.237,Z 79.749,A 180.000,B 0.000,C 180.000} C_DIS
LIN {X 96.474,Y 88.242,Z 79.747,A 180.000,B 0.000,C 180.000} C_DIS
LIN {X 96.399,Y 88.249,Z 79.744,A 180.000,B 0.000,C 180.000} C_DIS
LIN {X 96.325,Y 88.259,Z 79.742,A 180.000,B 0.000,C 180.000} C_DIS
LIN {X 96.102,Y 88.286,Z 79.734,A 180.000,B 0.000,C 180.000} C_DIS
LIN {X 96.028,Y 88.296,Z 79.731,A 180.000,B 0.000,C 180.000} C_DIS
LIN {X 95.954,Y 88.307,Z 79.729,A 180.000,B 0.000,C 180.000} C_DIS
LIN {X 95.881,Y 88.320,Z 79.726,A 180.000,B 0.000,C 180.000} C_DIS
LIN {X 95.804,Y 88.334,Z 79.723,A 180.000,B 0.000,C 180.000} C_DIS
LIN {X 95.727,Y 88.347,Z 79.720,A 180.000,B 0.000,C 180.000} C_DIS
LIN {X 95.499,Y 88.389,Z 79.712,A 180.000,B 0.000,C 180.000} C_DIS
LIN {X 95.426,Y 88.402,Z 79.710,A 180.000,B 0.000,C 180.000} C_DIS
LIN {X 95.354,Y 88.417,Z 79.707,A 180.000,B 0.000,C 180.000} C_DIS
LIN {X 95.281,Y 88.434,Z 79.705,A 180.000,B 0.000,C 180.000} C_DIS
LIN {X 95.134,Y 88.470,Z 79.699,A 180.000,B 0.000,C 180.000} C_DIS
LIN {X 95.060,Y 88.488,Z 79.697,A 180.000,B 0.000,C 180.000} C_DIS
LIN {X 94.987,Y 88.506,Z 79.694,A 180.000,B 0.000,C 180.000} C_DIS
LIN {X 94.912,Y 88.526,Z 79.691,A 180.000,B 0.000,C 180.000} C_DIS
LIN {X 94.839,Y 88.548,Z 79.689,A 180.000,B 0.000,C 180.000} C_DIS
LIN {X 94.617,Y 88.615,Z 79.681,A 180.000,B 0.000,C 180.000} C_DIS
LIN {X 94.543,Y 88.637,Z 79.678,A 180.000,B 0.000,C 180.000} C_DIS
LIN {X 94.469,Y 88.660,Z 79.675,A 180.000,B 0.000,C 180.000} C_DIS
LIN {X 94.395,Y 88.683,Z 79.672,A 180.000,B 0.000,C 180.000} C_DIS
LIN {X 94.323,Y 88.707,Z 79.670,A 180.000,B 0.000,C 180.000} C_DIS
LIN {X 94.252,Y 88.732,Z 79.667,A 180.000,B 0.000,C 180.000} C_DIS
LIN {X 94.039,Y 88.810,Z 79.659,A 180.000,B 0.000,C 180.000} C_DIS
LIN {X 93.968,Y 88.836,Z 79.657,A 180.000,B 0.000,C 180.000} C_DIS
LIN {X 93.898,Y 88.864,Z 79.654,A 180.000,B 0.000,C 180.000} C_DIS
LIN {X 93.828,Y 88.893,Z 79.651,A 180.000,B 0.000,C 180.000} C_DIS
LIN {X 93.616,Y 88.984,Z 79.643,A 180.000,B 0.000,C 180.000} C_DIS
LIN {X 93.546,Y 89.015,Z 79.641,A 180.000,B 0.000,C 180.000} C_DIS
LIN {X 93.408,Y 89.077,Z 79.635,A 180.000,B 0.000,C 180.000} C_DIS
LIN {X 93.339,Y 89.108,Z 79.633,A 180.000,B 0.000,C 180.000} C_DIS
LIN {X 93.272,Y 89.142,Z 79.630,A 180.000,B 0.000,C 180.000} C_DIS
LIN {X 93.061,Y 89.246,Z 79.622,A 180.000,B 0.000,C 180.000} C_DIS
LIN {X 92.991,Y 89.282,Z 79.619,A 180.000,B 0.000,C 180.000} C_DIS
LIN {X 92.925,Y 89.317,Z 79.616,A 180.000,B 0.000,C 180.000} C_DIS
LIN {X 92.859,Y 89.354,Z 79.614,A 180.000,B 0.000,C 180.000} C_DIS
LIN {X 92.662,Y 89.466,Z 79.606,A 180.000,B 0.000,C 180.000} C_DIS
LIN {X 92.596,Y 89.504,Z 79.603,A 180.000,B 0.000,C 180.000} C_DIS
LIN {X 92.531,Y 89.544,Z 79.601,A 180.000,B 0.000,C 180.000} C_DIS
LIN {X 92.466,Y 89.584,Z 79.598,A 180.000,B 0.000,C 180.000} C_DIS
LIN {X 92.400,Y 89.624,Z 79.595,A 180.000,B 0.000,C 180.000} C_DIS
LIN {X 92.335,Y 89.666,Z 79.593,A 180.000,B 0.000,C 180.000} C_DIS
LIN {X 92.142,Y 89.790,Z 79.585,A 180.000,B 0.000,C 180.000} C_DIS
LIN {X 92.079,Y 89.831,Z 79.582,A 180.000,B 0.000,C 180.000} C_DIS
LIN {X 92.017,Y 89.874,Z 79.579,A 180.000,B 0.000,C 180.000} C_DIS
LIN {X 91.956,Y 89.918,Z 79.577,A 180.000,B 0.000,C 180.000} C_DIS
LIN {X 91.766,Y 90.056,Z 79.568,A 180.000,B 0.000,C 180.000} C_DIS
LIN {X 91.703,Y 90.103,Z 79.566,A 180.000,B 0.000,C 180.000} C_DIS
LIN {X 91.644,Y 90.149,Z 79.563,A 180.000,B 0.000,C 180.000} C_DIS
LIN {X 91.526,Y 90.243,Z 79.558,A 180.000,B 0.000,C 180.000} C_DIS
LIN {X 91.468,Y 90.291,Z 79.555,A 180.000,B 0.000,C 180.000} C_DIS
LIN {X 91.289,Y 90.437,Z 79.547,A 180.000,B 0.000,C 180.000} C_DIS
LIN {X 91.230,Y 90.485,Z 79.544,A 180.000,B 0.000,C 180.000} C_DIS
LIN {X 91.172,Y 90.536,Z 79.542,A 180.000,B 0.000,C 180.000} C_DIS
LIN {X 91.115,Y 90.588,Z 79.539,A 180.000,B 0.000,C 180.000} C_DIS
LIN {X 90.945,Y 90.743,Z 79.531,A 180.000,B 0.000,C 180.000} C_DIS
LIN {X 90.890,Y 90.794,Z 79.528,A 180.000,B 0.000,C 180.000} C_DIS
LIN {X 90.836,Y 90.846,Z 79.526,A 180.000,B 0.000,C 180.000} C_DIS
LIN {X 90.784,Y 90.900,Z 79.523,A 180.000,B 0.000,C 180.000} C_DIS
LIN {X 90.619,Y 91.069,Z 79.515,A 180.000,B 0.000,C 180.000} C_DIS
LIN {X 90.564,Y 91.125,Z 79.512,A 180.000,B 0.000,C 180.000} C_DIS
LIN {X 90.511,Y 91.180,Z 79.510,A 180.000,B 0.000,C 180.000} C_DIS
LIN {X 90.459,Y 91.234,Z 79.507,A 180.000,B 0.000,C 180.000} C_DIS
LIN {X 90.408,Y 91.290,Z 79.504,A 180.000,B 0.000,C 180.000} C_DIS
LIN {X 90.358,Y 91.346,Z 79.502,A 180.000,B 0.000,C 180.000} C_DIS
LIN {X 90.205,Y 91.522,Z 79.493,A 180.000,B 0.000,C 180.000} C_DIS
LIN {X 90.154,Y 91.581,Z 79.491,A 180.000,B 0.000,C 180.000} C_DIS
LIN {X 90.105,Y 91.640,Z 79.488,A 180.000,B 0.000,C 180.000} C_DIS
LIN {X 90.058,Y 91.701,Z 79.485,A 180.000,B 0.000,C 180.000} C_DIS
LIN {X 89.917,Y 91.883,Z 79.477,A 180.000,B 0.000,C 180.000} C_DIS
LIN {X 89.870,Y 91.944,Z 79.475,A 180.000,B 0.000,C 180.000} C_DIS
LIN {X 89.776,Y 92.068,Z 79.469,A 180.000,B 0.000,C 180.000} C_DIS
LIN {X 89.731,Y 92.131,Z 79.467,A 180.000,B 0.000,C 180.000} C_DIS
LIN {X 89.687,Y 92.194,Z 79.464,A 180.000,B 0.000,C 180.000} C_DIS
LIN {X 89.556,Y 92.382,Z 79.456,A 180.000,B 0.000,C 180.000} C_DIS
LIN {X 89.514,Y 92.445,Z 79.453,A 180.000,B 0.000,C 180.000} C_DIS
LIN {X 89.473,Y 92.509,Z 79.451,A 180.000,B 0.000,C 180.000} C_DIS
LIN {X 89.433,Y 92.573,Z 79.448,A 180.000,B 0.000,C 180.000} C_DIS
LIN {X 89.310,Y 92.774,Z 79.440,A 180.000,B 0.000,C 180.000} C_DIS
LIN {X 89.270,Y 92.841,Z 79.437,A 180.000,B 0.000,C 180.000} C_DIS
LIN {X 89.232,Y 92.907,Z 79.434,A 180.000,B 0.000,C 180.000} C_DIS
LIN {X 89.194,Y 92.973,Z 79.432,A 180.000,B 0.000,C 180.000} C_DIS
LIN {X 89.157,Y 93.040,Z 79.429,A 180.000,B 0.000,C 180.000} C_DIS
LIN {X 89.120,Y 93.107,Z 79.426,A 180.000,B 0.000,C 180.000} C_DIS
LIN {X 89.009,Y 93.314,Z 79.418,A 180.000,B 0.000,C 180.000} C_DIS
LIN {X 88.972,Y 93.384,Z 79.415,A 180.000,B 0.000,C 180.000} C_DIS
LIN {X 88.938,Y 93.452,Z 79.413,A 180.000,B 0.000,C 180.000} C_DIS
LIN {X 88.906,Y 93.521,Z 79.410,A 180.000,B 0.000,C 180.000} C_DIS
LIN {X 88.809,Y 93.729,Z 79.402,A 180.000,B 0.000,C 180.000} C_DIS
LIN {X 88.777,Y 93.799,Z 79.399,A 180.000,B 0.000,C 180.000} C_DIS
LIN {X 88.747,Y 93.869,Z 79.397,A 180.000,B 0.000,C 180.000} C_DIS
LIN {X 88.688,Y 94.012,Z 79.391,A 180.000,B 0.000,C 180.000} C_DIS
LIN {X 88.659,Y 94.085,Z 79.389,A 180.000,B 0.000,C 180.000} C_DIS
LIN {X 88.572,Y 94.301,Z 79.380,A 180.000,B 0.000,C 180.000} C_DIS
LIN {X 88.544,Y 94.372,Z 79.378,A 180.000,B 0.000,C 180.000} C_DIS
LIN {X 88.518,Y 94.444,Z 79.375,A 180.000,B 0.000,C 180.000} C_DIS
LIN {X 88.493,Y 94.516,Z 79.372,A 180.000,B 0.000,C 180.000} C_DIS
LIN {X 88.420,Y 94.735,Z 79.364,A 180.000,B 0.000,C 180.000} C_DIS
LIN {X 88.396,Y 94.808,Z 79.362,A 180.000,B 0.000,C 180.000} C_DIS
LIN {X 88.374,Y 94.883,Z 79.359,A 180.000,B 0.000,C 180.000} C_DIS
LIN {X 88.353,Y 94.959,Z 79.356,A 180.000,B 0.000,C 180.000} C_DIS
LIN {X 88.290,Y 95.185,Z 79.348,A 180.000,B 0.000,C 180.000} C_DIS
LIN {X 88.270,Y 95.260,Z 79.345,A 180.000,B 0.000,C 180.000} C_DIS
LIN {X 88.249,Y 95.335,Z 79.343,A 180.000,B 0.000,C 180.000} C_DIS
LIN {X 88.229,Y 95.410,Z 79.340,A 180.000,B 0.000,C 180.000} C_DIS
LIN {X 88.211,Y 95.485,Z 79.337,A 180.000,B 0.000,C 180.000} C_DIS
LIN {X 88.195,Y 95.561,Z 79.334,A 180.000,B 0.000,C 180.000} C_DIS
LIN {X 88.146,Y 95.787,Z 79.326,A 180.000,B 0.000,C 180.000} C_DIS
LIN {X 88.130,Y 95.862,Z 79.324,A 180.000,B 0.000,C 180.000} C_DIS
LIN {X 88.117,Y 95.938,Z 79.321,A 180.000,B 0.000,C 180.000} C_DIS
LIN {X 88.105,Y 96.014,Z 79.318,A 180.000,B 0.000,C 180.000} C_DIS
LIN {X 88.080,Y 96.169,Z 79.313,A 180.000,B 0.000,C 180.000} C_DIS
LIN {X 88.068,Y 96.246,Z 79.310,A 180.000,B 0.000,C 180.000} C_DIS
LIN {X 88.056,Y 96.324,Z 79.307,A 180.000,B 0.000,C 180.000} C_DIS
LIN {X 88.046,Y 96.400,Z 79.305,A 180.000,B 0.000,C 180.000} C_DIS
LIN {X 88.035,Y 96.476,Z 79.302,A 180.000,B 0.000,C 180.000} C_DIS
LIN {X 88.025,Y 96.553,Z 79.299,A 180.000,B 0.000,C 180.000} C_DIS
LIN {X 88.017,Y 96.629,Z 79.297,A 180.000,B 0.000,C 180.000} C_DIS
LIN {X 88.002,Y 96.784,Z 79.291,A 180.000,B 0.000,C 180.000} C_DIS
LIN {X 87.994,Y 96.861,Z 79.288,A 180.000,B 0.000,C 180.000} C_DIS
LIN {X 87.987,Y 96.938,Z 79.286,A 180.000,B 0.000,C 180.000} C_DIS
LIN {X 87.982,Y 97.016,Z 79.283,A 180.000,B 0.000,C 180.000} C_DIS
LIN {X 87.978,Y 97.094,Z 79.280,A 180.000,B 0.000,C 180.000} C_DIS
LIN {X 87.968,Y 97.328,Z 79.272,A 180.000,B 0.000,C 180.000} C_DIS
LIN {X 87.965,Y 97.406,Z 79.269,A 180.000,B 0.000,C 180.000} C_DIS
LIN {X 87.964,Y 97.484,Z 79.267,A 180.000,B 0.000,C 180.000} C_DIS
LIN {X 87.963,Y 97.561,Z 79.264,A 180.000,B 0.000,C 180.000} C_DIS
LIN {X 87.962,Y 97.639,Z 79.261,A 180.000,B 0.000,C 180.000} C_DIS
LIN {X 87.963,Y 97.717,Z 79.259,A 180.000,B 0.000,C 180.000} C_DIS
LIN {X 87.966,Y 97.950,Z 79.250,A 180.000,B 0.000,C 180.000} C_DIS
LIN {X 87.967,Y 98.027,Z 79.248,A 180.000,B 0.000,C 180.000} C_DIS
LIN {X 87.971,Y 98.104,Z 79.245,A 180.000,B 0.000,C 180.000} C_DIS
LIN {X 87.976,Y 98.181,Z 79.242,A 180.000,B 0.000,C 180.000} C_DIS
LIN {X 87.987,Y 98.337,Z 79.237,A 180.000,B 0.000,C 180.000} C_DIS
LIN {X 87.992,Y 98.416,Z 79.234,A 180.000,B 0.000,C 180.000} C_DIS
LIN {X 87.998,Y 98.493,Z 79.231,A 180.000,B 0.000,C 180.000} C_DIS
LIN {X 88.006,Y 98.571,Z 79.229,A 180.000,B 0.000,C 180.000} C_DIS
LIN {X 88.015,Y 98.648,Z 79.226,A 180.000,B 0.000,C 180.000} C_DIS
LIN {X 88.023,Y 98.726,Z 79.223,A 180.000,B 0.000,C 180.000} C_DIS
LIN {X 88.033,Y 98.803,Z 79.221,A 180.000,B 0.000,C 180.000} C_DIS
LIN {X 88.052,Y 98.958,Z 79.215,A 180.000,B 0.000,C 180.000} C_DIS
LIN {X 88.062,Y 99.036,Z 79.212,A 180.000,B 0.000,C 180.000} C_DIS
LIN {X 88.072,Y 99.113,Z 79.210,A 180.000,B 0.000,C 180.000} C_DIS
LIN {X 88.084,Y 99.190,Z 79.207,A 180.000,B 0.000,C 180.000} C_DIS
LIN {X 88.098,Y 99.267,Z 79.204,A 180.000,B 0.000,C 180.000} C_DIS
LIN {X 88.140,Y 99.496,Z 79.196,A 180.000,B 0.000,C 180.000} C_DIS
LIN {X 88.155,Y 99.573,Z 79.193,A 180.000,B 0.000,C 180.000} C_DIS
LIN {X 88.172,Y 99.649,Z 79.191,A 180.000,B 0.000,C 180.000} C_DIS
LIN {X 88.208,Y 99.801,Z 79.185,A 180.000,B 0.000,C 180.000} C_DIS
LIN {X 88.227,Y 99.877,Z 79.182,A 180.000,B 0.000,C 180.000} C_DIS
LIN {X 88.245,Y 99.953,Z 79.180,A 180.000,B 0.000,C 180.000} C_DIS
LIN {X 88.263,Y 100.030,Z 79.177,A 180.000,B 0.000,C 180.000} C_DIS
LIN {X 88.282,Y 100.105,Z 79.175,A 180.000,B 0.000,C 180.000} C_DIS
LIN {X 88.300,Y 100.181,Z 79.172,A 180.000,B 0.000,C 180.000} C_DIS
LIN {X 88.321,Y 100.255,Z 79.169,A 180.000,B 0.000,C 180.000} C_DIS
LIN {X 88.344,Y 100.330,Z 79.167,A 180.000,B 0.000,C 180.000} C_DIS
LIN {X 88.366,Y 100.405,Z 79.164,A 180.000,B 0.000,C 180.000} C_DIS
LIN {X 88.389,Y 100.479,Z 79.162,A 180.000,B 0.000,C 180.000} C_DIS
LIN {X 88.412,Y 100.554,Z 79.159,A 180.000,B 0.000,C 180.000} C_DIS
LIN {X 88.435,Y 100.629,Z 79.157,A 180.000,B 0.000,C 180.000} C_DIS
LIN {X 88.461,Y 100.703,Z 79.154,A 180.000,B 0.000,C 180.000} C_DIS
LIN {X 88.487,Y 100.776,Z 79.151,A 180.000,B 0.000,C 180.000} C_DIS
LIN {X 88.541,Y 100.924,Z 79.147,A 180.000,B 0.000,C 180.000} C_DIS
LIN {X 88.595,Y 101.070,Z 79.142,A 180.000,B 0.000,C 180.000} C_DIS
LIN {X 88.651,Y 101.216,Z 79.137,A 180.000,B 0.000,C 180.000} C_DIS
LIN {X 88.712,Y 101.361,Z 79.132,A 180.000,B 0.000,C 180.000} C_DIS
LIN {X 88.774,Y 101.505,Z 79.127,A 180.000,B 0.000,C 180.000} C_DIS
LIN {X 88.836,Y 101.648,Z 79.123,A 180.000,B 0.000,C 180.000} C_DIS
LIN {X 88.905,Y 101.788,Z 79.118,A 180.000,B 0.000,C 180.000} C_DIS
LIN {X 88.975,Y 101.928,Z 79.114,A 180.000,B 0.000,C 180.000} C_DIS
LIN {X 89.046,Y 102.068,Z 79.109,A 180.000,B 0.000,C 180.000} C_DIS
LIN {X 89.119,Y 102.207,Z 79.105,A 180.000,B 0.000,C 180.000} C_DIS
LIN {X 89.196,Y 102.344,Z 79.100,A 180.000,B 0.000,C 180.000} C_DIS
LIN {X 89.274,Y 102.479,Z 79.096,A 180.000,B 0.000,C 180.000} C_DIS
LIN {X 89.352,Y 102.615,Z 79.092,A 180.000,B 0.000,C 180.000} C_DIS
LIN {X 89.437,Y 102.747,Z 79.088,A 180.000,B 0.000,C 180.000} C_DIS
LIN {X 89.523,Y 102.879,Z 79.084,A 180.000,B 0.000,C 180.000} C_DIS
LIN {X 89.609,Y 103.010,Z 79.080,A 180.000,B 0.000,C 180.000} C_DIS
LIN {X 89.699,Y 103.138,Z 79.076,A 180.000,B 0.000,C 180.000} C_DIS
LIN {X 89.792,Y 103.265,Z 79.072,A 180.000,B 0.000,C 180.000} C_DIS
LIN {X 89.885,Y 103.392,Z 79.069,A 180.000,B 0.000,C 180.000} C_DIS
LIN {X 89.979,Y 103.518,Z 79.065,A 180.000,B 0.000,C 180.000} C_DIS
LIN {X 90.078,Y 103.639,Z 79.062,A 180.000,B 0.000,C 180.000} C_DIS
LIN {X 90.178,Y 103.760,Z 79.058,A 180.000,B 0.000,C 180.000} C_DIS
LIN {X 90.278,Y 103.881,Z 79.055,A 180.000,B 0.000,C 180.000} C_DIS
LIN {X 90.384,Y 103.997,Z 79.052,A 180.000,B 0.000,C 180.000} C_DIS
LIN {X 90.491,Y 104.112,Z 79.048,A 180.000,B 0.000,C 180.000} C_DIS
LIN {X 90.598,Y 104.228,Z 79.045,A 180.000,B 0.000,C 180.000} C_DIS
LIN {X 90.705,Y 104.342,Z 79.042,A 180.000,B 0.000,C 180.000} C_DIS
LIN {X 90.818,Y 104.452,Z 79.039,A 180.000,B 0.000,C 180.000} C_DIS
LIN {X 90.931,Y 104.561,Z 79.037,A 180.000,B 0.000,C 180.000} C_DIS
LIN {X 91.045,Y 104.669,Z 79.034,A 180.000,B 0.000,C 180.000} C_DIS
LIN {X 91.164,Y 104.772,Z 79.031,A 180.000,B 0.000,C 180.000} C_DIS
LIN {X 91.403,Y 104.977,Z 79.026,A 180.000,B 0.000,C 180.000} C_DIS
LIN {X 91.648,Y 105.174,Z 79.022,A 180.000,B 0.000,C 180.000} C_DIS
LIN {X 91.899,Y 105.364,Z 79.018,A 180.000,B 0.000,C 180.000} C_DIS
LIN {X 92.159,Y 105.541,Z 79.014,A 180.000,B 0.000,C 180.000} C_DIS
LIN {X 92.423,Y 105.713,Z 79.011,A 180.000,B 0.000,C 180.000} C_DIS
LIN {X 92.693,Y 105.876,Z 79.008,A 180.000,B 0.000,C 180.000} C_DIS
LIN {X 92.967,Y 106.029,Z 79.005,A 180.000,B 0.000,C 180.000} C_DIS
LIN {X 93.247,Y 106.173,Z 79.003,A 180.000,B 0.000,C 180.000} C_DIS
LIN {X 93.533,Y 106.306,Z 79.002,A 180.000,B 0.000,C 180.000} C_DIS
LIN {X 93.821,Y 106.435,Z 79.001,A 180.000,B 0.000,C 180.000} C_DIS
LIN {X 94.114,Y 106.548,Z 79.000,A 180.000,B 0.000,C 180.000} C_DIS
LIN {X 94.321,Y 106.622,Z 79.000,A 180.000,B 0.000,C 180.000} C_DIS
; Cutting Move Starts
LIN {X 94.394,Y 106.647,Z 79.000,A 180.000,B 0.000,C 180.000} C_DIS
LIN {X 94.573,Y 106.704,Z 79.000,A 180.000,B 0.000,C 180.000} C_DIS
LIN {X 94.751,Y 106.761,Z 79.000,A 180.000,B 0.000,C 180.000} C_DIS
LIN {X 94.930,Y 106.814,Z 79.000,A 180.000,B 0.000,C 180.000} C_DIS
LIN {X 95.109,Y 106.860,Z 79.000,A 180.000,B 0.000,C 180.000} C_DIS
LIN {X 95.288,Y 106.906,Z 79.000,A 180.000,B 0.000,C 180.000} C_DIS
LIN {X 95.295,Y 106.908,Z 79.000,A 180.000,B 0.000,C 180.000} C_DIS
LIN {X 95.466,Y 106.943,Z 79.000,A 180.000,B 0.000,C 180.000} C_DIS
LIN {X 95.645,Y 106.979,Z 79.000,A 180.000,B 0.000,C 180.000} C_DIS
LIN {X 95.824,Y 107.014,Z 79.000,A 180.000,B 0.000,C 180.000} C_DIS
LIN {X 96.003,Y 107.045,Z 79.000,A 180.000,B 0.000,C 180.000} C_DIS
LIN {X 96.296,Y 107.086,Z 79.000,A 180.000,B 0.000,C 180.000} C_DIS
LIN {X 96.360,Y 107.095,Z 79.000,A 180.000,B 0.000,C 180.000} C_DIS
LIN {X 96.539,Y 107.113,Z 79.000,A 180.000,B 0.000,C 180.000} C_DIS
LIN {X 96.718,Y 107.128,Z 79.000,A 180.000,B 0.000,C 180.000} C_DIS
LIN {X 96.897,Y 107.141,Z 79.000,A 180.000,B 0.000,C 180.000} C_DIS
LIN {X 97.075,Y 107.152,Z 79.000,A 180.000,B 0.000,C 180.000} C_DIS
LIN {X 97.254,Y 107.157,Z 79.000,A 180.000,B 0.000,C 180.000} C_DIS
LIN {X 97.433,Y 107.162,Z 79.000,A 180.000,B 0.000,C 180.000} C_DIS
LIN {X 97.612,Y 107.161,Z 79.000,A 180.000,B 0.000,C 180.000} C_DIS
LIN {X 97.790,Y 107.156,Z 79.000,A 180.000,B 0.000,C 180.000} C_DIS
LIN {X 97.969,Y 107.150,Z 79.000,A 180.000,B 0.000,C 180.000} C_DIS
LIN {X 98.148,Y 107.139,Z 79.000,A 180.000,B 0.000,C 180.000} C_DIS
LIN {X 98.327,Y 107.124,Z 79.000,A 180.000,B 0.000,C 180.000} C_DIS
LIN {X 98.505,Y 107.109,Z 79.000,A 180.000,B 0.000,C 180.000} C_DIS
LIN {X 98.684,Y 107.089,Z 79.000,A 180.000,B 0.000,C 180.000} C_DIS
LIN {X 98.863,Y 107.064,Z 79.000,A 180.000,B 0.000,C 180.000} C_DIS
LIN {X 99.042,Y 107.038,Z 79.000,A 180.000,B 0.000,C 180.000} C_DIS
LIN {X 99.221,Y 107.005,Z 79.000,A 180.000,B 0.000,C 180.000} C_DIS
LIN {X 99.399,Y 106.970,Z 79.000,A 180.000,B 0.000,C 180.000} C_DIS
LIN {X 99.578,Y 106.935,Z 79.000,A 180.000,B 0.000,C 180.000} C_DIS
LIN {X 99.705,Y 106.908,Z 79.000,A 180.000,B 0.000,C 180.000} C_DIS
LIN {X 99.757,Y 106.895,Z 79.000,A 180.000,B 0.000,C 180.000} C_DIS
LIN {X 99.936,Y 106.849,Z 79.000,A 180.000,B 0.000,C 180.000} C_DIS
LIN {X 100.114,Y 106.802,Z 79.000,A 180.000,B 0.000,C 180.000} C_DIS
LIN {X 100.293,Y 106.747,Z 79.000,A 180.000,B 0.000,C 180.000} C_DIS
LIN {X 100.472,Y 106.690,Z 79.000,A 180.000,B 0.000,C 180.000} C_DIS
LIN {X 100.651,Y 106.632,Z 79.000,A 180.000,B 0.000,C 180.000} C_DIS
LIN {X 100.829,Y 106.570,Z 79.000,A 180.000,B 0.000,C 180.000} C_DIS
LIN {X 101.008,Y 106.501,Z 79.000,A 180.000,B 0.000,C 180.000} C_DIS
LIN {X 101.187,Y 106.432,Z 79.000,A 180.000,B 0.000,C 180.000} C_DIS
LIN {X 101.324,Y 106.371,Z 79.000,A 180.000,B 0.000,C 180.000} C_DIS
LIN {X 101.545,Y 106.273,Z 79.000,A 180.000,B 0.000,C 180.000} C_DIS
LIN {X 101.716,Y 106.193,Z 79.000,A 180.000,B 0.000,C 180.000} C_DIS
LIN {X 101.723,Y 106.189,Z 79.000,A 180.000,B 0.000,C 180.000} C_DIS
LIN {X 101.902,Y 106.099,Z 79.000,A 180.000,B 0.000,C 180.000} C_DIS
LIN {X 102.081,Y 106.007,Z 79.000,A 180.000,B 0.000,C 180.000} C_DIS
LIN {X 102.260,Y 105.908,Z 79.000,A 180.000,B 0.000,C 180.000} C_DIS
LIN {X 102.438,Y 105.803,Z 79.000,A 180.000,B 0.000,C 180.000} C_DIS
LIN {X 102.617,Y 105.694,Z 79.000,A 180.000,B 0.000,C 180.000} C_DIS
LIN {X 102.677,Y 105.656,Z 79.000,A 180.000,B 0.000,C 180.000} C_DIS
LIN {X 102.796,Y 105.579,Z 79.000,A 180.000,B 0.000,C 180.000} C_DIS
LIN {X 102.975,Y 105.460,Z 79.000,A 180.000,B 0.000,C 180.000} C_DIS
LIN {X 103.153,Y 105.336,Z 79.000,A 180.000,B 0.000,C 180.000} C_DIS
LIN {X 103.203,Y 105.299,Z 79.000,A 180.000,B 0.000,C 180.000} C_DIS
LIN {X 103.332,Y 105.201,Z 79.000,A 180.000,B 0.000,C 180.000} C_DIS
LIN {X 103.440,Y 105.120,Z 79.000,A 180.000,B 0.000,C 180.000} C_DIS
LIN {X 103.511,Y 105.064,Z 79.000,A 180.000,B 0.000,C 180.000} C_DIS
LIN {X 103.659,Y 104.941,Z 79.000,A 180.000,B 0.000,C 180.000} C_DIS
LIN {X 103.871,Y 104.762,Z 79.000,A 180.000,B 0.000,C 180.000} C_DIS
LIN {X 104.047,Y 104.605,Z 79.000,A 180.000,B 0.000,C 180.000} C_DIS
LIN {X 104.226,Y 104.436,Z 79.000,A 180.000,B 0.000,C 180.000} C_DIS
LIN {X 104.259,Y 104.405,Z 79.000,A 180.000,B 0.000,C 180.000} C_DIS
LIN {X 104.405,Y 104.255,Z 79.000,A 180.000,B 0.000,C 180.000} C_DIS
LIN {X 104.584,Y 104.066,Z 79.000,A 180.000,B 0.000,C 180.000} C_DIS
LIN {X 104.601,Y 104.047,Z 79.000,A 180.000,B 0.000,C 180.000} C_DIS
LIN {X 104.762,Y 103.873,Z 79.000,A 180.000,B 0.000,C 180.000} C_DIS
LIN {X 104.766,Y 103.869,Z 79.000,A 180.000,B 0.000,C 180.000} C_DIS
LIN {X 104.917,Y 103.690,Z 79.000,A 180.000,B 0.000,C 180.000} C_DIS
LIN {X 104.941,Y 103.662,Z 79.000,A 180.000,B 0.000,C 180.000} C_DIS
LIN {X 105.065,Y 103.511,Z 79.000,A 180.000,B 0.000,C 180.000} C_DIS
LIN {X 105.120,Y 103.439,Z 79.000,A 180.000,B 0.000,C 180.000} C_DIS
LIN {X 105.200,Y 103.332,Z 79.000,A 180.000,B 0.000,C 180.000} C_DIS
LIN {X 105.299,Y 103.201,Z 79.000,A 180.000,B 0.000,C 180.000} C_DIS
LIN {X 105.333,Y 103.153,Z 79.000,A 180.000,B 0.000,C 180.000} C_DIS
LIN {X 105.460,Y 102.975,Z 79.000,A 180.000,B 0.000,C 180.000} C_DIS
LIN {X 105.580,Y 102.796,Z 79.000,A 180.000,B 0.000,C 180.000} C_DIS
LIN {X 105.656,Y 102.681,Z 79.000,A 180.000,B 0.000,C 180.000} C_DIS
LIN {X 105.697,Y 102.617,Z 79.000,A 180.000,B 0.000,C 180.000} C_DIS
LIN {X 105.802,Y 102.438,Z 79.000,A 180.000,B 0.000,C 180.000} C_DIS
LIN {X 105.835,Y 102.383,Z 79.000,A 180.000,B 0.000,C 180.000} C_DIS
LIN {X 105.907,Y 102.260,Z 79.000,A 180.000,B 0.000,C 180.000} C_DIS
LIN {X 106.006,Y 102.081,Z 79.000,A 180.000,B 0.000,C 180.000} C_DIS
LIN {X 106.014,Y 102.066,Z 79.000,A 180.000,B 0.000,C 180.000} C_DIS
LIN {X 106.099,Y 101.902,Z 79.000,A 180.000,B 0.000,C 180.000} C_DIS
LIN {X 106.191,Y 101.723,Z 79.000,A 180.000,B 0.000,C 180.000} C_DIS
LIN {X 106.193,Y 101.720,Z 79.000,A 180.000,B 0.000,C 180.000} C_DIS
LIN {X 106.274,Y 101.545,Z 79.000,A 180.000,B 0.000,C 180.000} C_DIS
LIN {X 106.371,Y 101.327,Z 79.000,A 180.000,B 0.000,C 180.000} C_DIS
LIN {X 106.430,Y 101.187,Z 79.000,A 180.000,B 0.000,C 180.000} C_DIS
LIN {X 106.500,Y 101.008,Z 79.000,A 180.000,B 0.000,C 180.000} C_DIS
LIN {X 106.568,Y 100.829,Z 79.000,A 180.000,B 0.000,C 180.000} C_DIS
LIN {X 106.635,Y 100.651,Z 79.000,A 180.000,B 0.000,C 180.000} C_DIS
LIN {X 106.692,Y 100.472,Z 79.000,A 180.000,B 0.000,C 180.000} C_DIS
LIN {X 106.749,Y 100.293,Z 79.000,A 180.000,B 0.000,C 180.000} C_DIS
LIN {X 106.800,Y 100.114,Z 79.000,A 180.000,B 0.000,C 180.000} C_DIS
LIN {X 106.846,Y 99.936,Z 79.000,A 180.000,B 0.000,C 180.000} C_DIS
LIN {X 106.892,Y 99.757,Z 79.000,A 180.000,B 0.000,C 180.000} C_DIS
LIN {X 106.908,Y 99.696,Z 79.000,A 180.000,B 0.000,C 180.000} C_DIS
LIN {X 106.936,Y 99.578,Z 79.000,A 180.000,B 0.000,C 180.000} C_DIS
LIN {X 106.972,Y 99.399,Z 79.000,A 180.000,B 0.000,C 180.000} C_DIS
LIN {X 107.008,Y 99.221,Z 79.000,A 180.000,B 0.000,C 180.000} C_DIS
LIN {X 107.037,Y 99.042,Z 79.000,A 180.000,B 0.000,C 180.000} C_DIS
LIN {X 107.063,Y 98.863,Z 79.000,A 180.000,B 0.000,C 180.000} C_DIS
LIN {X 107.086,Y 98.689,Z 79.000,A 180.000,B 0.000,C 180.000} C_DIS
LIN {X 107.087,Y 98.684,Z 79.000,A 180.000,B 0.000,C 180.000} C_DIS
LIN {X 107.109,Y 98.505,Z 79.000,A 180.000,B 0.000,C 180.000} C_DIS
LIN {X 107.125,Y 98.327,Z 79.000,A 180.000,B 0.000,C 180.000} C_DIS
LIN {X 107.140,Y 98.148,Z 79.000,A 180.000,B 0.000,C 180.000} C_DIS
LIN {X 107.151,Y 97.969,Z 79.000,A 180.000,B 0.000,C 180.000} C_DIS
LIN {X 107.156,Y 97.790,Z 79.000,A 180.000,B 0.000,C 180.000} C_DIS
LIN {X 107.160,Y 97.612,Z 79.000,A 180.000,B 0.000,C 180.000} C_DIS
LIN {X 107.160,Y 97.433,Z 79.000,A 180.000,B 0.000,C 180.000} C_DIS
LIN {X 107.157,Y 97.254,Z 79.000,A 180.000,B 0.000,C 180.000} C_DIS
LIN {X 107.152,Y 97.075,Z 79.000,A 180.000,B 0.000,C 180.000} C_DIS
LIN {X 107.144,Y 96.897,Z 79.000,A 180.000,B 0.000,C 180.000} C_DIS
LIN {X 107.129,Y 96.718,Z 79.000,A 180.000,B 0.000,C 180.000} C_DIS
LIN {X 107.114,Y 96.539,Z 79.000,A 180.000,B 0.000,C 180.000} C_DIS
LIN {X 107.093,Y 96.360,Z 79.000,A 180.000,B 0.000,C 180.000} C_DIS
LIN {X 107.086,Y 96.311,Z 79.000,A 180.000,B 0.000,C 180.000} C_DIS
LIN {X 107.069,Y 96.181,Z 79.000,A 180.000,B 0.000,C 180.000} C_DIS
LIN {X 107.044,Y 96.003,Z 79.000,A 180.000,B 0.000,C 180.000} C_DIS
LIN {X 107.016,Y 95.824,Z 79.000,A 180.000,B 0.000,C 180.000} C_DIS
LIN {X 106.981,Y 95.645,Z 79.000,A 180.000,B 0.000,C 180.000} C_DIS
LIN {X 106.945,Y 95.466,Z 79.000,A 180.000,B 0.000,C 180.000} C_DIS
LIN {X 106.908,Y 95.304,Z 79.000,A 180.000,B 0.000,C 180.000} C_DIS
LIN {X 106.904,Y 95.288,Z 79.000,A 180.000,B 0.000,C 180.000} C_DIS
LIN {X 106.858,Y 95.109,Z 79.000,A 180.000,B 0.000,C 180.000} C_DIS
LIN {X 106.811,Y 94.930,Z 79.000,A 180.000,B 0.000,C 180.000} C_DIS
LIN {X 106.763,Y 94.751,Z 79.000,A 180.000,B 0.000,C 180.000} C_DIS
LIN {X 106.729,Y 94.643,Z 79.000,A 180.000,B 0.000,C 180.000} C_DIS
LIN {X 106.707,Y 94.573,Z 79.000,A 180.000,B 0.000,C 180.000} C_DIS
LIN {X 106.650,Y 94.394,Z 79.000,A 180.000,B 0.000,C 180.000} C_DIS
LIN {X 106.585,Y 94.215,Z 79.000,A 180.000,B 0.000,C 180.000} C_DIS
LIN {X 106.517,Y 94.036,Z 79.000,A 180.000,B 0.000,C 180.000} C_DIS
LIN {X 106.447,Y 93.857,Z 79.000,A 180.000,B 0.000,C 180.000} C_DIS
LIN {X 106.374,Y 93.679,Z 79.000,A 180.000,B 0.000,C 180.000} C_DIS
LIN {X 106.294,Y 93.500,Z 79.000,A 180.000,B 0.000,C 180.000} C_DIS
LIN {X 106.234,Y 93.369,Z 79.000,A 180.000,B 0.000,C 180.000} C_DIS
LIN {X 106.213,Y 93.321,Z 79.000,A 180.000,B 0.000,C 180.000} C_DIS
LIN {X 106.193,Y 93.280,Z 79.000,A 180.000,B 0.000,C 180.000} C_DIS
LIN {X 106.122,Y 93.142,Z 79.000,A 180.000,B 0.000,C 180.000} C_DIS
LIN {X 106.029,Y 92.964,Z 79.000,A 180.000,B 0.000,C 180.000} C_DIS
LIN {X 106.014,Y 92.934,Z 79.000,A 180.000,B 0.000,C 180.000} C_DIS
LIN {X 105.932,Y 92.785,Z 79.000,A 180.000,B 0.000,C 180.000} C_DIS
LIN {X 105.835,Y 92.617,Z 79.000,A 180.000,B 0.000,C 180.000} C_DIS
LIN {X 105.723,Y 92.427,Z 79.000,A 180.000,B 0.000,C 180.000} C_DIS
LIN {X 105.656,Y 92.319,Z 79.000,A 180.000,B 0.000,C 180.000} C_DIS
LIN {X 105.610,Y 92.249,Z 79.000,A 180.000,B 0.000,C 180.000} C_DIS
LIN {X 105.477,Y 92.051,Z 79.000,A 180.000,B 0.000,C 180.000} C_DIS
LIN {X 105.365,Y 91.891,Z 79.000,A 180.000,B 0.000,C 180.000} C_DIS
LIN {X 105.299,Y 91.799,Z 79.000,A 180.000,B 0.000,C 180.000} C_DIS
LIN {X 105.233,Y 91.712,Z 79.000,A 180.000,B 0.000,C 180.000} C_DIS
LIN {X 105.099,Y 91.533,Z 79.000,A 180.000,B 0.000,C 180.000} C_DIS
LIN {X 104.955,Y 91.355,Z 79.000,A 180.000,B 0.000,C 180.000} C_DIS
LIN {X 104.804,Y 91.176,Z 79.000,A 180.000,B 0.000,C 180.000} C_DIS
LIN {X 104.762,Y 91.127,Z 79.000,A 180.000,B 0.000,C 180.000} C_DIS
LIN {X 104.643,Y 90.997,Z 79.000,A 180.000,B 0.000,C 180.000} C_DIS
LIN {X 104.584,Y 90.934,Z 79.000,A 180.000,B 0.000,C 180.000} C_DIS
LIN {X 104.475,Y 90.818,Z 79.000,A 180.000,B 0.000,C 180.000} C_DIS
LIN {X 104.405,Y 90.745,Z 79.000,A 180.000,B 0.000,C 180.000} C_DIS
LIN {X 104.304,Y 90.640,Z 79.000,A 180.000,B 0.000,C 180.000} C_DIS
LIN {X 104.226,Y 90.564,Z 79.000,A 180.000,B 0.000,C 180.000} C_DIS
LIN {X 104.047,Y 90.395,Z 79.000,A 180.000,B 0.000,C 180.000} C_DIS
LIN {X 103.923,Y 90.282,Z 79.000,A 180.000,B 0.000,C 180.000} C_DIS
LIN {X 103.869,Y 90.236,Z 79.000,A 180.000,B 0.000,C 180.000} C_DIS
LIN {X 103.690,Y 90.085,Z 79.000,A 180.000,B 0.000,C 180.000} C_DIS
LIN {X 103.511,Y 89.936,Z 79.000,A 180.000,B 0.000,C 180.000} C_DIS
LIN {X 103.497,Y 89.925,Z 79.000,A 180.000,B 0.000,C 180.000} C_DIS
LIN {X 103.332,Y 89.799,Z 79.000,A 180.000,B 0.000,C 180.000} C_DIS
LIN {X 103.262,Y 89.746,Z 79.000,A 180.000,B 0.000,C 180.000} C_DIS
LIN {X 103.153,Y 89.664,Z 79.000,A 180.000,B 0.000,C 180.000} C_DIS
LIN {X 103.014,Y 89.567,Z 79.000,A 180.000,B 0.000,C 180.000} C_DIS
LIN {X 102.796,Y 89.421,Z 79.000,A 180.000,B 0.000,C 180.000} C_DIS
LIN {X 102.747,Y 89.388,Z 79.000,A 180.000,B 0.000,C 180.000} C_DIS
LIN {X 102.617,Y 89.306,Z 79.000,A 180.000,B 0.000,C 180.000} C_DIS
LIN {X 102.459,Y 89.209,Z 79.000,A 180.000,B 0.000,C 180.000} C_DIS
LIN {X 102.260,Y 89.092,Z 79.000,A 180.000,B 0.000,C 180.000} C_DIS
LIN {X 102.152,Y 89.031,Z 79.000,A 180.000,B 0.000,C 180.000} C_DIS
LIN {X 102.081,Y 88.993,Z 79.000,A 180.000,B 0.000,C 180.000} C_DIS
LIN {X 101.902,Y 88.901,Z 79.000,A 180.000,B 0.000,C 180.000} C_DIS
LIN {X 101.807,Y 88.852,Z 79.000,A 180.000,B 0.000,C 180.000} C_DIS
LIN {X 101.723,Y 88.811,Z 79.000,A 180.000,B 0.000,C 180.000} C_DIS
LIN {X 101.545,Y 88.727,Z 79.000,A 180.000,B 0.000,C 180.000} C_DIS
LIN {X 101.366,Y 88.647,Z 79.000,A 180.000,B 0.000,C 180.000} C_DIS
LIN {X 101.187,Y 88.568,Z 79.000,A 180.000,B 0.000,C 180.000} C_DIS
LIN {X 101.008,Y 88.499,Z 79.000,A 180.000,B 0.000,C 180.000} C_DIS
LIN {X 100.829,Y 88.430,Z 79.000,A 180.000,B 0.000,C 180.000} C_DIS
LIN {X 100.651,Y 88.368,Z 79.000,A 180.000,B 0.000,C 180.000} C_DIS
LIN {X 100.490,Y 88.316,Z 79.000,A 180.000,B 0.000,C 180.000} C_DIS
LIN {X 100.293,Y 88.253,Z 79.000,A 180.000,B 0.000,C 180.000} C_DIS
LIN {X 100.114,Y 88.198,Z 79.000,A 180.000,B 0.000,C 180.000} C_DIS
LIN {X 99.936,Y 88.151,Z 79.000,A 180.000,B 0.000,C 180.000} C_DIS
LIN {X 99.757,Y 88.105,Z 79.000,A 180.000,B 0.000,C 180.000} C_DIS
LIN {X 99.578,Y 88.065,Z 79.000,A 180.000,B 0.000,C 180.000} C_DIS
LIN {X 99.399,Y 88.030,Z 79.000,A 180.000,B 0.000,C 180.000} C_DIS
LIN {X 99.221,Y 87.995,Z 79.000,A 180.000,B 0.000,C 180.000} C_DIS
LIN {X 99.042,Y 87.962,Z 79.000,A 180.000,B 0.000,C 180.000} C_DIS
LIN {X 99.018,Y 87.958,Z 79.000,A 180.000,B 0.000,C 180.000} C_DIS
LIN {X 98.863,Y 87.936,Z 79.000,A 180.000,B 0.000,C 180.000} C_DIS
LIN {X 98.684,Y 87.911,Z 79.000,A 180.000,B 0.000,C 180.000} C_DIS
LIN {X 98.505,Y 87.891,Z 79.000,A 180.000,B 0.000,C 180.000} C_DIS
LIN {X 98.327,Y 87.876,Z 79.000,A 180.000,B 0.000,C 180.000} C_DIS
LIN {X 98.148,Y 87.861,Z 79.000,A 180.000,B 0.000,C 180.000} C_DIS
LIN {X 97.969,Y 87.850,Z 79.000,A 180.000,B 0.000,C 180.000} C_DIS
LIN {X 97.790,Y 87.844,Z 79.000,A 180.000,B 0.000,C 180.000} C_DIS
LIN {X 97.612,Y 87.839,Z 79.000,A 180.000,B 0.000,C 180.000} C_DIS
LIN {X 97.433,Y 87.838,Z 79.000,A 180.000,B 0.000,C 180.000} C_DIS
LIN {X 97.254,Y 87.843,Z 79.000,A 180.000,B 0.000,C 180.000} C_DIS
LIN {X 97.075,Y 87.848,Z 79.000,A 180.000,B 0.000,C 180.000} C_DIS
LIN {X 96.897,Y 87.859,Z 79.000,A 180.000,B 0.000,C 180.000} C_DIS
LIN {X 96.718,Y 87.872,Z 79.000,A 180.000,B 0.000,C 180.000} C_DIS
LIN {X 96.539,Y 87.887,Z 79.000,A 180.000,B 0.000,C 180.000} C_DIS
LIN {X 96.360,Y 87.905,Z 79.000,A 180.000,B 0.000,C 180.000} C_DIS
LIN {X 96.181,Y 87.930,Z 79.000,A 180.000,B 0.000,C 180.000} C_DIS
LIN {X 96.003,Y 87.955,Z 79.000,A 180.000,B 0.000,C 180.000} C_DIS
LIN {X 95.982,Y 87.958,Z 79.000,A 180.000,B 0.000,C 180.000} C_DIS
LIN {X 95.824,Y 87.986,Z 79.000,A 180.000,B 0.000,C 180.000} C_DIS
LIN {X 95.645,Y 88.021,Z 79.000,A 180.000,B 0.000,C 180.000} C_DIS
LIN {X 95.466,Y 88.057,Z 79.000,A 180.000,B 0.000,C 180.000} C_DIS
LIN {X 95.288,Y 88.094,Z 79.000,A 180.000,B 0.000,C 180.000} C_DIS
LIN {X 95.120,Y 88.137,Z 79.000,A 180.000,B 0.000,C 180.000} C_DIS
LIN {X 94.930,Y 88.186,Z 79.000,A 180.000,B 0.000,C 180.000} C_DIS
LIN {X 94.751,Y 88.239,Z 79.000,A 180.000,B 0.000,C 180.000} C_DIS
LIN {X 94.510,Y 88.316,Z 79.000,A 180.000,B 0.000,C 180.000} C_DIS
LIN {X 94.394,Y 88.353,Z 79.000,A 180.000,B 0.000,C 180.000} C_DIS
LIN {X 94.215,Y 88.413,Z 79.000,A 180.000,B 0.000,C 180.000} C_DIS
LIN {X 94.036,Y 88.482,Z 79.000,A 180.000,B 0.000,C 180.000} C_DIS
LIN {X 94.003,Y 88.494,Z 79.000,A 180.000,B 0.000,C 180.000} C_DIS
LIN {X 93.857,Y 88.550,Z 79.000,A 180.000,B 0.000,C 180.000} C_DIS
LIN {X 93.679,Y 88.627,Z 79.000,A 180.000,B 0.000,C 180.000} C_DIS
LIN {X 93.500,Y 88.707,Z 79.000,A 180.000,B 0.000,C 180.000} C_DIS
LIN {X 93.321,Y 88.790,Z 79.000,A 180.000,B 0.000,C 180.000} C_DIS
LIN {X 93.193,Y 88.852,Z 79.000,A 180.000,B 0.000,C 180.000} C_DIS
LIN {X 93.142,Y 88.878,Z 79.000,A 180.000,B 0.000,C 180.000} C_DIS
LIN {X 92.964,Y 88.970,Z 79.000,A 180.000,B 0.000,C 180.000} C_DIS
LIN {X 92.848,Y 89.031,Z 79.000,A 180.000,B 0.000,C 180.000} C_DIS
LIN {X 92.785,Y 89.066,Z 79.000,A 180.000,B 0.000,C 180.000} C_DIS
LIN {X 92.606,Y 89.171,Z 79.000,A 180.000,B 0.000,C 180.000} C_DIS
LIN {X 92.541,Y 89.209,Z 79.000,A 180.000,B 0.000,C 180.000} C_DIS
LIN {X 92.427,Y 89.278,Z 79.000,A 180.000,B 0.000,C 180.000} C_DIS
LIN {X 92.253,Y 89.388,Z 79.000,A 180.000,B 0.000,C 180.000} C_DIS
LIN {X 92.249,Y 89.391,Z 79.000,A 180.000,B 0.000,C 180.000} C_DIS
LIN {X 92.070,Y 89.511,Z 79.000,A 180.000,B 0.000,C 180.000} C_DIS
LIN {X 91.986,Y 89.567,Z 79.000,A 180.000,B 0.000,C 180.000} C_DIS
LIN {X 91.891,Y 89.632,Z 79.000,A 180.000,B 0.000,C 180.000} C_DIS
LIN {X 91.738,Y 89.746,Z 79.000,A 180.000,B 0.000,C 180.000} C_DIS
LIN {X 91.712,Y 89.765,Z 79.000,A 180.000,B 0.000,C 180.000} C_DIS
LIN {X 91.533,Y 89.900,Z 79.000,A 180.000,B 0.000,C 180.000} C_DIS
LIN {X 91.503,Y 89.925,Z 79.000,A 180.000,B 0.000,C 180.000} C_DIS
LIN {X 91.355,Y 90.047,Z 79.000,A 180.000,B 0.000,C 180.000} C_DIS
LIN {X 91.288,Y 90.103,Z 79.000,A 180.000,B 0.000,C 180.000} C_DIS
LIN {X 91.176,Y 90.198,Z 79.000,A 180.000,B 0.000,C 180.000} C_DIS
LIN {X 91.077,Y 90.282,Z 79.000,A 180.000,B 0.000,C 180.000} C_DIS
LIN {X 90.997,Y 90.353,Z 79.000,A 180.000,B 0.000,C 180.000} C_DIS
LIN {X 90.883,Y 90.461,Z 79.000,A 180.000,B 0.000,C 180.000} C_DIS
LIN {X 90.818,Y 90.522,Z 79.000,A 180.000,B 0.000,C 180.000} C_DIS
LIN {X 90.696,Y 90.640,Z 79.000,A 180.000,B 0.000,C 180.000} C_DIS
LIN {X 90.640,Y 90.698,Z 79.000,A 180.000,B 0.000,C 180.000} C_DIS
LIN {X 90.461,Y 90.887,Z 79.000,A 180.000,B 0.000,C 180.000} C_DIS
LIN {X 90.357,Y 90.997,Z 79.000,A 180.000,B 0.000,C 180.000} C_DIS
LIN {X 90.282,Y 91.077,Z 79.000,A 180.000,B 0.000,C 180.000} C_DIS
LIN {X 90.196,Y 91.176,Z 79.000,A 180.000,B 0.000,C 180.000} C_DIS
LIN {X 90.045,Y 91.355,Z 79.000,A 180.000,B 0.000,C 180.000} C_DIS
LIN {X 89.925,Y 91.502,Z 79.000,A 180.000,B 0.000,C 180.000} C_DIS
LIN {X 89.901,Y 91.533,Z 79.000,A 180.000,B 0.000,C 180.000} C_DIS
LIN {X 89.746,Y 91.740,Z 79.000,A 180.000,B 0.000,C 180.000} C_DIS
LIN {X 89.635,Y 91.891,Z 79.000,A 180.000,B 0.000,C 180.000} C_DIS
LIN {X 89.567,Y 91.985,Z 79.000,A 180.000,B 0.000,C 180.000} C_DIS
LIN {X 89.510,Y 92.070,Z 79.000,A 180.000,B 0.000,C 180.000} C_DIS
LIN {X 89.388,Y 92.252,Z 79.000,A 180.000,B 0.000,C 180.000} C_DIS
LIN {X 89.277,Y 92.427,Z 79.000,A 180.000,B 0.000,C 180.000} C_DIS
LIN {X 89.171,Y 92.606,Z 79.000,A 180.000,B 0.000,C 180.000} C_DIS
LIN {X 89.068,Y 92.785,Z 79.000,A 180.000,B 0.000,C 180.000} C_DIS
LIN {X 89.031,Y 92.853,Z 79.000,A 180.000,B 0.000,C 180.000} C_DIS
LIN {X 88.971,Y 92.964,Z 79.000,A 180.000,B 0.000,C 180.000} C_DIS
LIN {X 88.852,Y 93.194,Z 79.000,A 180.000,B 0.000,C 180.000} C_DIS
LIN {X 88.787,Y 93.321,Z 79.000,A 180.000,B 0.000,C 180.000} C_DIS
LIN {X 88.706,Y 93.500,Z 79.000,A 180.000,B 0.000,C 180.000} C_DIS
LIN {X 88.626,Y 93.679,Z 79.000,A 180.000,B 0.000,C 180.000} C_DIS
LIN {X 88.553,Y 93.857,Z 79.000,A 180.000,B 0.000,C 180.000} C_DIS
LIN {X 88.494,Y 94.007,Z 79.000,A 180.000,B 0.000,C 180.000} C_DIS
LIN {X 88.415,Y 94.215,Z 79.000,A 180.000,B 0.000,C 180.000} C_DIS
LIN {X 88.350,Y 94.394,Z 79.000,A 180.000,B 0.000,C 180.000} C_DIS
LIN {X 88.316,Y 94.503,Z 79.000,A 180.000,B 0.000,C 180.000} C_DIS
LIN {X 88.293,Y 94.573,Z 79.000,A 180.000,B 0.000,C 180.000} C_DIS
LIN {X 88.237,Y 94.751,Z 79.000,A 180.000,B 0.000,C 180.000} C_DIS
LIN {X 88.189,Y 94.930,Z 79.000,A 180.000,B 0.000,C 180.000} C_DIS
LIN {X 88.137,Y 95.131,Z 79.000,A 180.000,B 0.000,C 180.000} C_DIS
LIN {X 88.096,Y 95.288,Z 79.000,A 180.000,B 0.000,C 180.000} C_DIS
LIN {X 88.055,Y 95.466,Z 79.000,A 180.000,B 0.000,C 180.000} C_DIS
LIN {X 88.019,Y 95.645,Z 79.000,A 180.000,B 0.000,C 180.000} C_DIS
LIN {X 87.984,Y 95.824,Z 79.000,A 180.000,B 0.000,C 180.000} C_DIS
LIN {X 87.958,Y 95.991,Z 79.000,A 180.000,B 0.000,C 180.000} C_DIS
LIN {X 87.931,Y 96.181,Z 79.000,A 180.000,B 0.000,C 180.000} C_DIS
LIN {X 87.907,Y 96.360,Z 79.000,A 180.000,B 0.000,C 180.000} C_DIS
LIN {X 87.886,Y 96.539,Z 79.000,A 180.000,B 0.000,C 180.000} C_DIS
LIN {X 87.871,Y 96.718,Z 79.000,A 180.000,B 0.000,C 180.000} C_DIS
LIN {X 87.856,Y 96.897,Z 79.000,A 180.000,B 0.000,C 180.000} C_DIS
LIN {X 87.848,Y 97.075,Z 79.000,A 180.000,B 0.000,C 180.000} C_DIS
LIN {X 87.843,Y 97.254,Z 79.000,A 180.000,B 0.000,C 180.000} C_DIS
LIN {X 87.840,Y 97.433,Z 79.000,A 180.000,B 0.000,C 180.000} C_DIS
LIN {X 87.840,Y 97.612,Z 79.000,A 180.000,B 0.000,C 180.000} C_DIS
LIN {X 87.844,Y 97.790,Z 79.000,A 180.000,B 0.000,C 180.000} C_DIS
LIN {X 87.849,Y 97.969,Z 79.000,A 180.000,B 0.000,C 180.000} C_DIS
LIN {X 87.860,Y 98.148,Z 79.000,A 180.000,B 0.000,C 180.000} C_DIS
LIN {X 87.875,Y 98.327,Z 79.000,A 180.000,B 0.000,C 180.000} C_DIS
LIN {X 87.891,Y 98.505,Z 79.000,A 180.000,B 0.000,C 180.000} C_DIS
LIN {X 87.913,Y 98.684,Z 79.000,A 180.000,B 0.000,C 180.000} C_DIS
LIN {X 87.937,Y 98.863,Z 79.000,A 180.000,B 0.000,C 180.000} C_DIS
LIN {X 87.963,Y 99.042,Z 79.000,A 180.000,B 0.000,C 180.000} C_DIS
LIN {X 87.992,Y 99.221,Z 79.000,A 180.000,B 0.000,C 180.000} C_DIS
LIN {X 88.028,Y 99.399,Z 79.000,A 180.000,B 0.000,C 180.000} C_DIS
LIN {X 88.064,Y 99.578,Z 79.000,A 180.000,B 0.000,C 180.000} C_DIS
LIN {X 88.108,Y 99.757,Z 79.000,A 180.000,B 0.000,C 180.000} C_DIS
LIN {X 88.137,Y 99.869,Z 79.000,A 180.000,B 0.000,C 180.000} C_DIS
LIN {X 88.200,Y 100.114,Z 79.000,A 180.000,B 0.000,C 180.000} C_DIS
LIN {X 88.251,Y 100.293,Z 79.000,A 180.000,B 0.000,C 180.000} C_DIS
LIN {X 88.316,Y 100.497,Z 79.000,A 180.000,B 0.000,C 180.000} C_DIS
LIN {X 88.365,Y 100.651,Z 79.000,A 180.000,B 0.000,C 180.000} C_DIS
LIN {X 88.432,Y 100.829,Z 79.000,A 180.000,B 0.000,C 180.000} C_DIS
LIN {X 88.500,Y 101.008,Z 79.000,A 180.000,B 0.000,C 180.000} C_DIS
LIN {X 88.570,Y 101.187,Z 79.000,A 180.000,B 0.000,C 180.000} C_DIS
LIN {X 88.646,Y 101.366,Z 79.000,A 180.000,B 0.000,C 180.000} C_DIS
LIN {X 88.726,Y 101.545,Z 79.000,A 180.000,B 0.000,C 180.000} C_DIS
LIN {X 88.809,Y 101.723,Z 79.000,A 180.000,B 0.000,C 180.000} C_DIS
LIN {X 88.852,Y 101.806,Z 79.000,A 180.000,B 0.000,C 180.000} C_DIS
LIN {X 88.901,Y 101.902,Z 79.000,A 180.000,B 0.000,C 180.000} C_DIS
LIN {X 88.994,Y 102.081,Z 79.000,A 180.000,B 0.000,C 180.000} C_DIS
LIN {X 89.031,Y 102.147,Z 79.000,A 180.000,B 0.000,C 180.000} C_DIS
LIN {X 89.093,Y 102.260,Z 79.000,A 180.000,B 0.000,C 180.000} C_DIS
LIN {X 89.198,Y 102.438,Z 79.000,A 180.000,B 0.000,C 180.000} C_DIS
LIN {X 89.209,Y 102.459,Z 79.000,A 180.000,B 0.000,C 180.000} C_DIS
LIN {X 89.303,Y 102.617,Z 79.000,A 180.000,B 0.000,C 180.000} C_DIS
LIN {X 89.388,Y 102.748,Z 79.000,A 180.000,B 0.000,C 180.000} C_DIS
LIN {X 89.540,Y 102.975,Z 79.000,A 180.000,B 0.000,C 180.000} C_DIS
LIN {X 89.567,Y 103.015,Z 79.000,A 180.000,B 0.000,C 180.000} C_DIS
LIN {X 89.667,Y 103.153,Z 79.000,A 180.000,B 0.000,C 180.000} C_DIS
LIN {X 89.746,Y 103.260,Z 79.000,A 180.000,B 0.000,C 180.000} C_DIS
LIN {X 89.800,Y 103.332,Z 79.000,A 180.000,B 0.000,C 180.000} C_DIS
LIN {X 89.925,Y 103.498,Z 79.000,A 180.000,B 0.000,C 180.000} C_DIS
LIN {X 89.935,Y 103.511,Z 79.000,A 180.000,B 0.000,C 180.000} C_DIS
LIN {X 90.083,Y 103.690,Z 79.000,A 180.000,B 0.000,C 180.000} C_DIS
LIN {X 90.103,Y 103.714,Z 79.000,A 180.000,B 0.000,C 180.000} C_DIS
LIN {X 90.234,Y 103.869,Z 79.000,A 180.000,B 0.000,C 180.000} C_DIS
LIN {X 90.282,Y 103.923,Z 79.000,A 180.000,B 0.000,C 180.000} C_DIS
LIN {X 90.399,Y 104.047,Z 79.000,A 180.000,B 0.000,C 180.000} C_DIS
LIN {X 90.461,Y 104.113,Z 79.000,A 180.000,B 0.000,C 180.000} C_DIS
LIN {X 90.640,Y 104.302,Z 79.000,A 180.000,B 0.000,C 180.000} C_DIS
LIN {X 90.741,Y 104.405,Z 79.000,A 180.000,B 0.000,C 180.000} C_DIS
LIN {X 90.818,Y 104.478,Z 79.000,A 180.000,B 0.000,C 180.000} C_DIS
LIN {X 90.930,Y 104.584,Z 79.000,A 180.000,B 0.000,C 180.000} C_DIS
LIN {X 90.997,Y 104.647,Z 79.000,A 180.000,B 0.000,C 180.000} C_DIS
LIN {X 91.129,Y 104.762,Z 79.000,A 180.000,B 0.000,C 180.000} C_DIS
